C09115=1110.868,346.804,-84.343,-177.299,10.930,149.499
C09116=1110.872,346.556,-84.309,-177.302,10.928,149.499
C09117=1110.876,346.309,-84.274,-177.305,10.925,149.499
C09118=1110.880,346.062,-84.238,-177.308,10.923,149.499
C09119=1110.883,345.813,-84.203,-177.312,10.920,149.500
C09120=1110.888,345.567,-84.168,-177.314,10.918,149.500
C09121=1110.892,345.318,-84.133,-177.317,10.916,149.500
C09122=1110.895,345.071,-84.098,-177.321,10.913,149.500
C09123=1110.899,344.824,-84.064,-177.324,10.911,149.500
C09124=1110.903,344.576,-84.028,-177.327,10.908,149.501
C09125=1110.907,344.328,-83.994,-177.330,10.906,149.501
C09126=1110.911,344.081,-83.959,-177.334,10.903,149.501
C09127=1110.914,343.834,-83.924,-177.337,10.901,149.501
C09128=1110.919,343.586,-83.890,-177.340,10.898,149.501
C09129=1110.923,343.339,-83.854,-177.343,10.897,149.502
C09130=1110.927,343.091,-83.819,-177.346,10.894,149.502
C09131=1110.930,342.843,-83.785,-177.349,10.891,149.502
C09132=1110.934,342.596,-83.750,-177.352,10.889,149.502
C09133=1110.939,342.349,-83.715,-177.356,10.886,149.502
C09134=1110.943,342.100,-83.681,-177.359,10.884,149.503
C09135=1110.945,341.853,-83.646,-177.362,10.881,149.503
C09136=1110.950,341.606,-83.611,-177.365,10.879,149.503
C09137=1110.954,341.358,-83.576,-177.369,10.876,149.503
C09138=1110.958,341.111,-83.543,-177.372,10.874,149.503
C09139=1110.962,340.863,-83.507,-177.374,10.872,149.503
C09140=1110.966,340.616,-83.473,-177.378,10.869,149.504
C09141=1110.969,340.368,-83.438,-177.381,10.867,149.504
C09142=1110.974,340.120,-83.404,-177.384,10.864,149.504
C09143=1110.978,339.873,-83.368,-177.387,10.862,149.504
C09144=1110.981,339.625,-83.334,-177.390,10.859,149.504
C09145=1110.985,339.378,-83.300,-177.394,10.857,149.505
C09146=1110.989,339.130,-83.265,-177.397,10.854,149.505
C09147=1110.993,338.882,-83.231,-177.400,10.852,149.505
C09148=1110.997,338.634,-83.196,-177.403,10.849,149.505
C09149=1111.002,338.387,-83.162,-177.407,10.847,149.505
C09150=1111.005,338.139,-83.127,-177.409,10.845,149.506
C09151=1111.009,337.892,-83.092,-177.413,10.842,149.506
C09152=1111.012,337.645,-83.058,-177.415,10.840,149.506
C09153=1111.016,337.433,-83.029,-177.419,10.837,149.506
C09154=1111.019,337.221,-82.999,-177.421,10.835,149.506
C09155=1111.023,337.009,-82.970,-177.424,10.833,149.507
C09156=1111.026,336.797,-82.940,-177.427,10.831,149.507
C09157=1111.030,336.585,-82.911,-177.429,10.829,149.507
C09158=1111.034,336.373,-82.881,-177.432,10.827,149.507
C09159=1111.037,336.161,-82.852,-177.435,10.825,149.507
C09160=1111.039,335.949,-82.823,-177.437,10.823,149.507
C09161=1111.044,335.702,-82.788,-177.441,10.820,149.508
C09162=1111.047,335.454,-82.754,-177.444,10.818,149.508
C09163=1111.052,335.206,-82.720,-177.447,10.815,149.508
C09164=1111.056,334.959,-82.686,-177.450,10.812,149.508
C09165=1111.060,334.710,-82.652,-177.453,10.811,149.508
C09166=1111.063,334.463,-82.618,-177.456,10.808,149.509
C09167=1111.067,334.215,-82.583,-177.459,10.806,149.509
C09168=1111.071,333.968,-82.549,-177.462,10.803,149.509
C09169=1111.075,333.720,-82.515,-177.466,10.801,149.509
C09170=1111.079,333.473,-82.480,-177.469,10.798,149.509
C09171=1111.083,333.225,-82.447,-177.472,10.795,149.509
C09172=1111.087,332.977,-82.412,-177.475,10.793,149.510
C09173=1111.091,332.730,-82.379,-177.479,10.790,149.510
C09174=1111.094,332.482,-82.344,-177.481,10.788,149.510
C09175=1111.099,332.234,-82.311,-177.484,10.786,149.510
C09176=1111.103,331.987,-82.277,-177.487,10.784,149.510
C09177=1111.106,331.739,-82.242,-177.490,10.781,149.510
C09178=1111.111,331.492,-82.208,-177.494,10.778,149.511
C09179=1111.115,331.244,-82.175,-177.497,10.776,149.511
C09180=1111.118,330.996,-82.141,-177.500,10.773,149.511
C09181=1111.123,330.749,-82.106,-177.503,10.771,149.511
C09182=1111.127,330.501,-82.073,-177.507,10.768,149.512
C09183=1111.130,330.253,-82.039,-177.510,10.766,149.512
C09184=1111.134,330.006,-82.005,-177.513,10.763,149.512
C09185=1111.139,329.758,-81.971,-177.516,10.761,149.512
C09186=1111.142,329.510,-81.937,-177.519,10.759,149.512
C09187=1111.146,329.263,-81.904,-177.522,10.756,149.512
C09188=1111.150,329.015,-81.870,-177.525,10.754,149.513
C09189=1111.154,328.767,-81.836,-177.528,10.751,149.513
C09190=1111.158,328.520,-81.802,-177.531,10.748,149.513
C09191=1111.162,328.272,-81.768,-177.535,10.746,149.513
C09192=1111.165,328.024,-81.734,-177.538,10.743,149.513
C09193=1111.170,327.777,-81.700,-177.541,10.741,149.513
C09194=1111.174,327.529,-81.667,-177.544,10.738,149.514
C09195=1111.178,327.282,-81.633,-177.547,10.737,149.514
C09196=1111.182,327.033,-81.599,-177.550,10.734,149.514
C09197=1111.186,326.786,-81.566,-177.553,10.731,149.514
C09198=1111.190,326.539,-81.532,-177.556,10.729,149.515
C09199=1111.194,326.290,-81.499,-177.559,10.726,149.515
C09200=1111.198,326.043,-81.464,-177.563,10.724,149.515
C09201=1111.202,325.795,-81.431,-177.566,10.721,149.515
C09202=1111.206,325.547,-81.398,-177.569,10.718,149.515
C09203=1111.210,325.300,-81.364,-177.572,10.716,149.515
C09204=1111.213,325.052,-81.331,-177.576,10.714,149.516
C09205=1111.217,324.804,-81.298,-177.578,10.712,149.516
C09206=1111.221,324.557,-81.264,-177.581,10.709,149.516
C09207=1111.225,324.309,-81.231,-177.585,10.707,149.516
C09208=1111.230,324.061,-81.197,-177.587,10.704,149.516
C09209=1111.233,323.849,-81.168,-177.591,10.701,149.517
C09210=1111.237,323.637,-81.139,-177.593,10.699,149.517
C09211=1111.240,323.424,-81.111,-177.596,10.698,149.517
C09212=1111.243,323.213,-81.082,-177.599,10.695,149.517
C09213=1111.246,323.000,-81.053,-177.601,10.693,149.517
C09214=1111.250,322.788,-81.025,-177.604,10.691,149.517
C09215=1111.253,322.577,-80.996,-177.607,10.689,149.517
C09216=1111.256,322.364,-80.968,-177.609,10.687,149.518
C09217=1111.260,322.117,-80.935,-177.612,10.684,149.518
C09218=1111.264,321.869,-80.902,-177.616,10.682,149.518
C09219=1111.269,321.621,-80.869,-177.618,10.679,149.518
C09220=1111.272,321.374,-80.835,-177.621,10.677,149.518
C09221=1111.276,321.126,-80.801,-177.624,10.675,149.519
C09222=1111.280,320.878,-80.768,-177.627,10.672,149.519
C09223=1111.284,320.630,-80.735,-177.631,10.670,149.519
C09224=1111.288,320.382,-80.702,-177.634,10.667,149.519
C09225=1111.293,320.135,-80.668,-177.637,10.664,149.519
C09226=1111.297,319.887,-80.635,-177.640,10.662,149.519
C09227=1111.301,319.639,-80.602,-177.643,10.659,149.520
C09228=1111.304,319.391,-80.569,-177.647,10.657,149.520
C09229=1111.308,319.143,-80.536,-177.650,10.654,149.520
C09230=1111.312,318.896,-80.503,-177.652,10.652,149.520
C09231=1111.316,318.648,-80.470,-177.656,10.650,149.520
C09232=1111.320,318.400,-80.437,-177.658,10.647,149.520
C09233=1111.324,318.152,-80.403,-177.662,10.645,149.521
C09234=1111.328,317.905,-80.370,-177.665,10.642,149.521
C09235=1111.333,317.657,-80.337,-177.668,10.639,149.521
C09236=1111.336,317.410,-80.305,-177.671,10.637,149.521
C09237=1111.340,317.162,-80.271,-177.674,10.634,149.521
C09238=1111.344,316.914,-80.238,-177.678,10.632,149.522
C09239=1111.348,316.666,-80.205,-177.681,10.629,149.522
C09240=1111.353,316.418,-80.173,-177.683,10.627,149.522
C09241=1111.356,316.171,-80.140,-177.687,10.625,149.522
C09242=1111.360,315.922,-80.107,-177.689,10.622,149.522
C09243=1111.364,315.674,-80.073,-177.693,10.620,149.522
C09244=1111.368,315.427,-80.040,-177.696,10.617,149.523
C09245=1111.372,315.178,-80.008,-177.699,10.614,149.523
C09246=1111.376,314.931,-79.975,-177.702,10.612,149.523
C09247=1111.380,314.683,-79.942,-177.705,10.609,149.523
C09248=1111.384,314.436,-79.909,-177.709,10.607,149.523
C09249=1111.388,314.187,-79.877,-177.712,10.604,149.524
C09250=1111.392,313.940,-79.844,-177.714,10.602,149.524
C09251=1111.396,313.692,-79.811,-177.718,10.600,149.524
C09252=1111.400,313.444,-79.778,-177.720,10.597,149.524
C09253=1111.404,313.196,-79.746,-177.724,10.595,149.524
C09254=1111.408,312.949,-79.713,-177.727,10.592,149.524
C09255=1111.413,312.701,-79.681,-177.730,10.589,149.525
C09256=1111.417,312.453,-79.648,-177.733,10.587,149.525
C09257=1111.421,312.206,-79.615,-177.736,10.584,149.525
C09258=1111.424,311.958,-79.583,-177.740,10.582,149.525
C09259=1111.429,311.710,-79.550,-177.743,10.579,149.525
C09260=1111.433,311.462,-79.517,-177.745,10.577,149.526
C09261=1111.436,311.214,-79.485,-177.748,10.575,149.526
C09262=1111.441,310.966,-79.452,-177.752,10.572,149.526
C09263=1111.445,310.718,-79.419,-177.754,10.569,149.526
C09264=1111.448,310.471,-79.387,-177.758,10.567,149.526
C09265=1111.452,310.258,-79.360,-177.760,10.565,149.526
C09266=1111.455,310.046,-79.332,-177.763,10.562,149.527
C09267=1111.460,309.834,-79.303,-177.766,10.560,149.527
C09268=1111.463,309.621,-79.276,-177.768,10.558,149.527
C09269=1111.466,309.409,-79.248,-177.771,10.556,149.527
C09270=1111.469,309.197,-79.220,-177.774,10.554,149.527
C09271=1111.473,308.985,-79.192,-177.776,10.552,149.527
C09272=1111.476,308.773,-79.165,-177.779,10.550,149.528
C09273=1111.481,308.525,-79.132,-177.782,10.547,149.528
C09274=1111.484,308.277,-79.100,-177.786,10.544,149.528
C09275=1111.489,308.029,-79.067,-177.788,10.542,149.528
C09276=1111.492,307.781,-79.035,-177.791,10.540,149.528
C09277=1111.497,307.533,-79.002,-177.794,10.537,149.528
C09278=1111.501,307.286,-78.971,-177.797,10.535,149.529
C09279=1111.505,307.037,-78.938,-177.800,10.532,149.529
C09280=1111.509,306.790,-78.906,-177.804,10.530,149.529
C09281=1111.512,306.542,-78.874,-177.807,10.527,149.529
C09282=1111.517,306.294,-78.841,-177.810,10.524,149.529
C09283=1111.521,306.046,-78.810,-177.813,10.522,149.529
C09284=1111.525,305.798,-78.777,-177.816,10.520,149.530
C09285=1111.529,305.550,-78.745,-177.819,10.517,149.530
C09286=1111.534,305.302,-78.712,-177.822,10.515,149.530
C09287=1111.537,305.054,-78.681,-177.825,10.512,149.530
C09288=1111.541,304.807,-78.648,-177.828,10.510,149.530
C09289=1111.546,304.559,-78.616,-177.831,10.507,149.531
C09290=1111.549,304.311,-78.584,-177.834,10.504,149.531
C09291=1111.554,304.063,-78.552,-177.838,10.502,149.531
C09292=1111.558,303.815,-78.520,-177.841,10.499,149.531
C09293=1111.562,303.567,-78.488,-177.844,10.497,149.531
C09294=1111.566,303.319,-78.456,-177.846,10.495,149.531
C09295=1111.570,303.071,-78.424,-177.850,10.492,149.532
C09296=1111.574,302.824,-78.392,-177.852,10.489,149.532
C09297=1111.578,302.576,-78.359,-177.856,10.487,149.532
C09298=1111.582,302.328,-78.328,-177.859,10.484,149.532
C09299=1111.586,302.080,-78.296,-177.862,10.482,149.532
C09300=1111.591,301.832,-78.264,-177.865,10.479,149.532
C09301=1111.595,301.584,-78.232,-177.868,10.477,149.533
C09302=1111.598,301.336,-78.200,-177.871,10.474,149.533
C09303=1111.603,301.088,-78.168,-177.874,10.472,149.533
C09304=1111.607,300.840,-78.136,-177.877,10.469,149.533
C09305=1111.611,300.592,-78.104,-177.880,10.467,149.533
C09306=1111.615,300.345,-78.073,-177.883,10.464,149.533
C09307=1111.620,300.096,-78.041,-177.887,10.462,149.534
C09308=1111.624,299.848,-78.009,-177.889,10.459,149.534
C09309=1111.628,299.601,-77.978,-177.893,10.457,149.534
C09310=1111.632,299.353,-77.946,-177.896,10.454,149.534
C09311=1111.635,299.104,-77.914,-177.899,10.451,149.534
C09312=1111.640,298.857,-77.882,-177.902,10.449,149.534
C09313=1111.644,298.609,-77.850,-177.905,10.447,149.535
C09314=1111.648,298.361,-77.818,-177.908,10.444,149.535
C09315=1111.652,298.113,-77.787,-177.911,10.442,149.535
C09316=1111.656,297.865,-77.756,-177.914,10.439,149.535
C09317=1111.660,297.617,-77.724,-177.917,10.437,149.535
C09318=1111.665,297.369,-77.692,-177.920,10.434,149.535
C09319=1111.669,297.120,-77.661,-177.923,10.431,149.536
C09320=1111.673,296.872,-77.629,-177.926,10.429,149.536
C09321=1111.676,296.660,-77.601,-177.929,10.427,149.536
C09322=1111.680,296.448,-77.575,-177.931,10.425,149.536
C09323=1111.683,296.236,-77.548,-177.934,10.422,149.536
C09324=1111.687,296.023,-77.521,-177.937,10.420,149.536
C09325=1111.690,295.811,-77.494,-177.939,10.418,149.537
C09326=1111.694,295.599,-77.467,-177.942,10.416,149.537
C09327=1111.697,295.386,-77.440,-177.945,10.414,149.537
C09328=1111.700,295.174,-77.413,-177.947,10.412,149.537
C09329=1111.705,294.926,-77.381,-177.950,10.409,149.537
C09330=1111.709,294.678,-77.350,-177.953,10.407,149.537
C09331=1111.713,294.430,-77.318,-177.956,10.404,149.538
C09332=1111.718,294.182,-77.287,-177.959,10.401,149.538
C09333=1111.721,293.934,-77.256,-177.963,10.399,149.538
C09334=1111.725,293.686,-77.224,-177.966,10.396,149.538
C09335=1111.730,293.438,-77.193,-177.969,10.394,149.538
C09336=1111.733,293.190,-77.162,-177.971,10.392,149.538
C09337=1111.737,292.942,-77.131,-177.974,10.389,149.539
C09338=1111.741,292.694,-77.099,-177.978,10.387,149.539
C09339=1111.746,292.446,-77.068,-177.981,10.384,149.539
C09340=1111.749,292.198,-77.036,-177.984,10.381,149.539
C09341=1111.754,291.950,-77.006,-177.987,10.379,149.539
C09342=1111.758,291.702,-76.974,-177.990,10.376,149.540
C09343=1111.762,291.454,-76.943,-177.993,10.373,149.540
C09344=1111.766,291.206,-76.911,-177.996,10.372,149.540
C09345=1111.771,290.958,-76.880,-177.999,10.369,149.540
C09346=1111.775,290.709,-76.849,-178.002,10.367,149.540
C09347=1111.779,290.462,-76.818,-178.005,10.364,149.540
C09348=1111.782,290.214,-76.787,-178.008,10.361,149.540
C09349=1111.787,289.966,-76.756,-178.011,10.359,149.541
C09350=1111.791,289.718,-76.725,-178.014,10.356,149.541
C09351=1111.795,289.470,-76.694,-178.018,10.354,149.541
C09352=1111.799,289.222,-76.662,-178.020,10.351,149.541
C09353=1111.804,288.974,-76.631,-178.023,10.349,149.542
C09354=1111.807,288.726,-76.601,-178.026,10.346,149.542
C09355=1111.811,288.478,-76.570,-178.029,10.344,149.542
C09356=1111.816,288.230,-76.539,-178.032,10.341,149.542
C09357=1111.820,287.982,-76.507,-178.035,10.338,149.542
C09358=1111.824,287.734,-76.477,-178.039,10.336,149.542
C09359=1111.828,287.485,-76.446,-178.042,10.333,149.542
C09360=1111.832,287.238,-76.415,-178.045,10.331,149.543
C09361=1111.836,286.989,-76.384,-178.048,10.328,149.543
C09362=1111.841,286.741,-76.353,-178.051,10.326,149.543
C09363=1111.844,286.494,-76.323,-178.053,10.324,149.543
C09364=1111.848,286.245,-76.291,-178.056,10.321,149.543
C09365=1111.853,285.997,-76.261,-178.060,10.318,149.544
C09366=1111.857,285.750,-76.229,-178.063,10.316,149.544
C09367=1111.861,285.501,-76.199,-178.066,10.313,149.544
C09368=1111.865,285.253,-76.168,-178.069,10.310,149.544
C09369=1111.869,285.005,-76.137,-178.072,10.308,149.544
C09370=1111.873,284.757,-76.107,-178.075,10.306,149.544
C09371=1111.878,284.509,-76.076,-178.078,10.303,149.544
C09372=1111.882,284.260,-76.045,-178.081,10.301,149.545
C09373=1111.886,284.013,-76.014,-178.084,10.298,149.545
C09374=1111.890,283.765,-75.984,-178.087,10.296,149.545
C09375=1111.894,283.516,-75.953,-178.090,10.293,149.545
C09376=1111.898,283.269,-75.922,-178.093,10.290,149.545
C09377=1111.902,283.055,-75.896,-178.096,10.289,149.546
C09378=1111.906,282.844,-75.870,-178.098,10.287,149.546
C09379=1111.909,282.631,-75.844,-178.101,10.284,149.546
C09380=1111.913,282.418,-75.817,-178.103,10.282,149.546
C09381=1111.916,282.206,-75.791,-178.106,10.280,149.546
C09382=1111.920,281.994,-75.765,-178.109,10.277,149.546
C09383=1111.924,281.781,-75.739,-178.111,10.275,149.546
C09384=1111.927,281.568,-75.713,-178.114,10.273,149.547
C09385=1111.932,281.320,-75.682,-178.117,10.271,149.547
C09386=1111.935,281.072,-75.652,-178.120,10.268,149.547
C09387=1111.939,280.824,-75.621,-178.123,10.265,149.547
C09388=1111.943,280.576,-75.591,-178.126,10.263,149.547
C09389=1111.948,280.328,-75.560,-178.129,10.260,149.547
C09390=1111.952,280.080,-75.530,-178.132,10.258,149.548
C09391=1111.956,279.831,-75.499,-178.135,10.255,149.548
C09392=1111.960,279.584,-75.469,-178.138,10.252,149.548
C09393=1111.965,279.336,-75.438,-178.142,10.250,149.548
C09394=1111.969,279.087,-75.409,-178.145,10.247,149.548
C09395=1111.973,278.839,-75.378,-178.147,10.244,149.548
C09396=1111.977,278.591,-75.348,-178.151,10.242,149.549
C09397=1111.981,278.343,-75.317,-178.154,10.239,149.549
C09398=1111.986,278.095,-75.287,-178.157,10.236,149.549
C09399=1111.990,277.847,-75.257,-178.159,10.234,149.549
C09400=1111.993,277.598,-75.226,-178.162,10.232,149.549
C09401=1111.998,277.350,-75.197,-178.165,10.229,149.549
C09402=1112.002,277.102,-75.166,-178.168,10.227,149.549
C09403=1112.006,276.855,-75.136,-178.171,10.224,149.550
C09404=1112.011,276.606,-75.106,-178.174,10.221,149.550
C09405=1112.014,276.358,-75.075,-178.177,10.219,149.550
C09406=1112.018,276.109,-75.046,-178.180,10.216,149.550
C09407=1112.023,275.861,-75.015,-178.183,10.213,149.550
C09408=1112.027,275.614,-74.985,-178.186,10.210,149.550
C09409=1112.031,275.366,-74.955,-178.189,10.208,149.550
C09410=1112.036,275.118,-74.924,-178.192,10.205,149.550
C09411=1112.039,274.869,-74.895,-178.195,10.203,149.551
C09412=1112.043,274.621,-74.864,-178.198,10.200,149.551
C09413=1112.048,274.372,-74.834,-178.201,10.198,149.551
C09414=1112.052,274.125,-74.804,-178.204,10.195,149.551
C09415=1112.056,273.876,-74.775,-178.207,10.192,149.551
C09416=1112.061,273.628,-74.744,-178.209,10.189,149.551
C09417=1112.065,273.380,-74.715,-178.212,10.187,149.551
C09418=1112.069,273.132,-74.685,-178.215,10.184,149.551
C09419=1112.073,272.884,-74.655,-178.218,10.182,149.551
C09420=1112.077,272.635,-74.625,-178.221,10.179,149.552
C09421=1112.081,272.387,-74.594,-178.224,10.177,149.552
C09422=1112.085,272.139,-74.565,-178.227,10.174,149.552
C09423=1112.090,271.891,-74.535,-178.230,10.171,149.552
C09424=1112.094,271.643,-74.505,-178.233,10.168,149.552
C09425=1112.098,271.395,-74.475,-178.236,10.166,149.552
C09426=1112.103,271.146,-74.446,-178.238,10.164,149.552
C09427=1112.106,270.899,-74.416,-178.241,10.161,149.552
C09428=1112.111,270.650,-74.386,-178.244,10.158,149.553
C09429=1112.116,270.402,-74.356,-178.247,10.155,149.553
C09430=1112.120,270.154,-74.327,-178.250,10.153,149.553
C09431=1112.124,269.906,-74.297,-178.252,10.151,149.553
C09432=1112.128,269.658,-74.267,-178.255,10.148,149.553
C09433=1112.131,269.445,-74.241,-178.257,10.146,149.553
C09434=1112.135,269.232,-74.216,-178.260,10.143,149.553
C09435=1112.138,269.019,-74.190,-178.263,10.141,149.553
C09436=1112.143,268.807,-74.166,-178.265,10.139,149.553
C09437=1112.146,268.594,-74.140,-178.267,10.137,149.553
C09438=1112.150,268.382,-74.114,-178.270,10.134,149.554
C09439=1112.153,268.168,-74.089,-178.272,10.132,149.554
C09440=1112.157,267.956,-74.064,-178.274,10.130,149.554
C09441=1112.161,267.708,-74.034,-178.277,10.127,149.554
C09442=1112.165,267.460,-74.005,-178.280,10.125,149.554
C09443=1112.170,267.211,-73.975,-178.282,10.123,149.554
C09444=1112.174,266.963,-73.946,-178.285,10.120,149.554
C09445=1112.178,266.715,-73.916,-178.288,10.117,149.554
C09446=1112.182,266.467,-73.886,-178.291,10.115,149.554
C09447=1112.186,266.219,-73.857,-178.294,10.112,149.555
C09448=1112.190,265.971,-73.827,-178.297,10.110,149.555
C09449=1112.194,265.723,-73.798,-178.299,10.107,149.555
C09450=1112.199,265.474,-73.768,-178.302,10.105,149.555
C09451=1112.203,265.226,-73.739,-178.305,10.102,149.555
C09452=1112.207,264.978,-73.709,-178.308,10.100,149.555
C09453=1112.211,264.729,-73.680,-178.310,10.098,149.555
C09454=1112.215,264.481,-73.650,-178.313,10.095,149.555
C09455=1112.220,264.232,-73.622,-178.316,10.092,149.556
C09456=1112.224,263.984,-73.592,-178.319,10.089,149.556
C09457=1112.229,263.736,-73.563,-178.323,10.087,149.556
C09458=1112.233,263.488,-73.534,-178.326,10.084,149.556
C09459=1112.237,263.240,-73.504,-178.328,10.081,149.556
C09460=1112.241,262.992,-73.475,-178.331,10.079,149.556
C09461=1112.246,262.743,-73.445,-178.334,10.076,149.556
C09462=1112.250,262.495,-73.416,-178.338,10.074,149.557
C09463=1112.254,262.247,-73.386,-178.341,10.071,149.557
C09464=1112.258,261.998,-73.358,-178.344,10.068,149.557
C09465=1112.262,261.751,-73.329,-178.346,10.065,149.557
C09466=1112.267,261.502,-73.300,-178.349,10.063,149.557
C09467=1112.271,261.254,-73.270,-178.352,10.060,149.557
C09468=1112.275,261.006,-73.241,-178.355,10.057,149.557
C09469=1112.279,260.757,-73.212,-178.358,10.054,149.557
C09470=1112.284,260.509,-73.183,-178.361,10.051,149.558
C09471=1112.288,260.261,-73.154,-178.364,10.049,149.558
C09472=1112.292,260.013,-73.125,-178.367,10.046,149.558
C09473=1112.296,259.764,-73.096,-178.370,10.043,149.558
C09474=1112.301,259.516,-73.067,-178.373,10.040,149.558
C09475=1112.305,259.267,-73.038,-178.375,10.037,149.558
C09476=1112.309,259.019,-73.008,-178.378,10.035,149.558
C09477=1112.313,258.772,-72.980,-178.381,10.032,149.558
C09478=1112.318,258.523,-72.951,-178.384,10.029,149.558
C09479=1112.322,258.275,-72.922,-178.387,10.026,149.558
C09480=1112.326,258.026,-72.892,-178.390,10.023,149.558
C09481=1112.330,257.778,-72.864,-178.393,10.020,149.558
C09482=1112.335,257.530,-72.835,-178.396,10.018,149.558
C09483=1112.339,257.281,-72.806,-178.398,10.016,149.559
C09484=1112.343,257.033,-72.777,-178.400,10.013,149.558
C09485=1112.347,256.784,-72.749,-178.403,10.010,149.559
C09486=1112.352,256.537,-72.720,-178.406,10.007,149.559
C09487=1112.356,256.288,-72.691,-178.409,10.004,149.559
C09488=1112.360,256.040,-72.662,-178.412,10.001,149.559
C09489=1112.364,255.827,-72.637,-178.413,10.000,149.559
C09490=1112.367,255.615,-72.613,-178.415,9.997,149.559
C09491=1112.371,255.401,-72.588,-178.417,9.996,149.559
C09492=1112.375,255.189,-72.563,-178.419,9.994,149.559
C09493=1112.379,254.976,-72.539,-178.420,9.992,149.559
C09494=1112.382,254.763,-72.514,-178.422,9.990,149.559
C09495=1112.386,254.551,-72.489,-178.424,9.988,149.559
C09496=1112.390,254.338,-72.464,-178.426,9.987,149.559
C09497=1112.393,254.089,-72.436,-178.429,9.984,149.559
C09498=1112.398,253.841,-72.407,-178.431,9.982,149.559
C09499=1112.403,253.593,-72.379,-178.433,9.980,149.559
C09500=1112.406,253.344,-72.350,-178.436,9.977,149.559
C09501=1112.411,253.096,-72.321,-178.438,9.975,149.559
C09502=1112.415,252.848,-72.293,-178.440,9.973,149.559
C09503=1112.419,252.599,-72.264,-178.444,9.971,149.560
C09504=1112.424,252.351,-72.235,-178.447,9.968,149.560
C09505=1112.428,252.103,-72.207,-178.449,9.966,149.560
C09506=1112.432,251.854,-72.178,-178.452,9.963,149.560
C09507=1112.436,251.606,-72.150,-178.455,9.961,149.560
C09508=1112.441,251.358,-72.121,-178.458,9.958,149.561
C09509=1112.445,251.109,-72.093,-178.461,9.955,149.561
C09510=1112.449,250.861,-72.064,-178.465,9.953,149.561
C09511=1112.453,250.613,-72.036,-178.467,9.950,149.561
C09512=1112.458,250.364,-72.007,-178.471,9.948,149.561
C09513=1112.462,250.116,-71.979,-178.474,9.945,149.561
C09514=1112.467,249.868,-71.951,-178.477,9.941,149.562
C09515=1112.470,249.620,-71.922,-178.481,9.939,149.562
C09516=1112.475,249.371,-71.893,-178.484,9.935,149.562
C09517=1112.479,249.123,-71.865,-178.488,9.933,149.562
C09518=1112.483,248.874,-71.836,-178.491,9.929,149.562
C09519=1112.488,248.626,-71.809,-178.495,9.926,149.563
C09520=1112.491,248.378,-71.781,-178.499,9.923,149.563
C09521=1112.497,248.129,-71.752,-178.502,9.919,149.563
C09522=1112.500,247.881,-71.724,-178.506,9.916,149.563
C09523=1112.505,247.633,-71.696,-178.510,9.913,149.563
C09524=1112.509,247.384,-71.668,-178.512,9.909,149.563
C09525=1112.513,247.135,-71.639,-178.515,9.906,149.563
C09526=1112.518,246.887,-71.611,-178.517,9.904,149.563
C09527=1112.522,246.639,-71.583,-178.519,9.901,149.563
C09528=1112.526,246.391,-71.555,-178.521,9.899,149.563
C09529=1112.531,246.142,-71.526,-178.524,9.896,149.563
C09530=1112.535,245.894,-71.499,-178.526,9.893,149.563
C09531=1112.539,245.645,-71.470,-178.529,9.890,149.563
C09532=1112.544,245.397,-71.442,-178.531,9.888,149.563
C09533=1112.548,245.149,-71.414,-178.533,9.885,149.563
C09534=1112.552,244.901,-71.386,-178.535,9.883,149.563
C09535=1112.556,244.652,-71.357,-178.538,9.880,149.563
C09536=1112.561,244.404,-71.330,-178.540,9.877,149.563
C09537=1112.564,244.156,-71.301,-178.543,9.875,149.563
C09538=1112.570,243.907,-71.274,-178.545,9.872,149.563
C09539=1112.574,243.658,-71.246,-178.547,9.869,149.563
C09540=1112.578,243.410,-71.218,-178.549,9.867,149.563
C09541=1112.582,243.162,-71.190,-178.552,9.864,149.563
C09542=1112.587,242.913,-71.161,-178.554,9.862,149.563
C09543=1112.591,242.665,-71.133,-178.557,9.859,149.563
C09544=1112.595,242.416,-71.106,-178.559,9.857,149.563
C09545=1112.599,242.204,-71.082,-178.561,9.855,149.563
C09546=1112.602,241.991,-71.058,-178.563,9.853,149.563
C09547=1112.607,241.778,-71.034,-178.565,9.850,149.563
C09548=1112.610,241.565,-71.010,-178.568,9.849,149.563
C09549=1112.613,241.352,-70.986,-178.570,9.845,149.563
C09550=1112.617,241.139,-70.962,-178.572,9.843,149.563
C09551=1112.621,240.926,-70.939,-178.574,9.841,149.563
C09552=1112.624,240.713,-70.915,-178.577,9.839,149.563
C09553=1112.629,240.465,-70.887,-178.579,9.837,149.563
C09554=1112.633,240.216,-70.859,-178.581,9.834,149.563
C09555=1112.638,239.968,-70.831,-178.584,9.831,149.563
C09556=1112.642,239.720,-70.804,-178.587,9.829,149.564
C09557=1112.646,239.471,-70.776,-178.589,9.826,149.563
C09558=1112.651,239.223,-70.748,-178.592,9.824,149.564
C09559=1112.654,238.974,-70.720,-178.595,9.821,149.564
C09560=1112.660,238.726,-70.693,-178.597,9.819,149.564
C09561=1112.664,238.478,-70.665,-178.599,9.816,149.564
C09562=1112.668,238.229,-70.637,-178.602,9.814,149.564
C09563=1112.672,237.981,-70.610,-178.605,9.811,149.564
C09564=1112.677,237.733,-70.582,-178.608,9.809,149.564
C09565=1112.681,237.483,-70.554,-178.610,9.806,149.564
C09566=1112.685,237.236,-70.527,-178.613,9.803,149.564
C09567=1112.689,236.986,-70.499,-178.615,9.801,149.564
C09568=1112.694,236.739,-70.472,-178.618,9.798,149.564
C09569=1112.698,236.490,-70.444,-178.621,9.796,149.565
C09570=1112.702,236.241,-70.416,-178.624,9.792,149.565
C09571=1112.707,235.993,-70.389,-178.626,9.790,149.565
C09572=1112.711,235.745,-70.361,-178.629,9.788,149.565
C09573=1112.716,235.497,-70.334,-178.632,9.785,149.565
C09574=1112.719,235.248,-70.306,-178.635,9.782,149.565
C09575=1112.724,235.000,-70.279,-178.637,9.780,149.565
C09576=1112.729,234.751,-70.252,-178.640,9.777,149.565
C09577=1112.732,234.502,-70.224,-178.643,9.774,149.565
C09578=1112.737,234.254,-70.197,-178.646,9.772,149.565
C09579=1112.742,234.005,-70.170,-178.649,9.769,149.565
C09580=1112.746,233.757,-70.142,-178.652,9.766,149.566
C09581=1112.750,233.508,-70.115,-178.654,9.763,149.566
C09582=1112.755,233.261,-70.087,-178.656,9.761,149.566
C09583=1112.759,233.012,-70.060,-178.659,9.758,149.566
C09584=1112.763,232.763,-70.032,-178.662,9.756,149.566
C09585=1112.768,232.514,-70.005,-178.665,9.752,149.566
C09586=1112.772,232.267,-69.978,-178.668,9.750,149.566
C09587=1112.776,232.018,-69.951,-178.671,9.747,149.566
C09588=1112.780,231.769,-69.924,-178.674,9.744,149.566
C09589=1112.785,231.521,-69.897,-178.676,9.741,149.566
C09590=1112.789,231.273,-69.869,-178.679,9.738,149.566
C09591=1112.794,231.024,-69.842,-178.682,9.736,149.566
C09592=1112.798,230.775,-69.814,-178.685,9.733,149.566
C09593=1112.802,230.527,-69.788,-178.688,9.730,149.566
C09594=1112.807,230.278,-69.761,-178.690,9.727,149.567
C09595=1112.811,230.030,-69.734,-178.693,9.724,149.567
C09596=1112.816,229.782,-69.706,-178.696,9.721,149.567
C09597=1112.820,229.533,-69.679,-178.700,9.718,149.567
C09598=1112.824,229.285,-69.652,-178.702,9.715,149.567
C09599=1112.828,229.036,-69.625,-178.705,9.712,149.567
C09600=1112.833,228.788,-69.598,-178.708,9.709,149.567
C09601=1112.837,228.575,-69.574,-178.710,9.707,149.567
C09602=1112.841,228.361,-69.552,-178.712,9.704,149.567
C09603=1112.844,228.148,-69.529,-178.715,9.702,149.567
C09604=1112.847,227.935,-69.505,-178.717,9.698,149.567
C09605=1112.852,227.723,-69.482,-178.719,9.696,149.567
C09606=1112.856,227.509,-69.459,-178.722,9.693,149.567
C09607=1112.859,227.296,-69.436,-178.724,9.691,149.567
C09608=1112.862,227.084,-69.413,-178.726,9.688,149.567
C09609=1112.867,226.835,-69.386,-178.729,9.685,149.567
C09610=1112.872,226.587,-69.359,-178.732,9.682,149.567
C09611=1112.876,226.338,-69.332,-178.734,9.679,149.567
C09612=1112.880,226.089,-69.306,-178.737,9.676,149.567
C09613=1112.885,225.840,-69.279,-178.739,9.673,149.567
C09614=1112.889,225.592,-69.252,-178.742,9.670,149.567
C09615=1112.893,225.343,-69.225,-178.745,9.667,149.567
C09616=1112.898,225.095,-69.198,-178.747,9.664,149.567
C09617=1112.902,224.847,-69.171,-178.750,9.661,149.567
C09618=1112.906,224.598,-69.144,-178.753,9.658,149.567
C09619=1112.911,224.350,-69.117,-178.755,9.654,149.566
C09620=1112.915,224.101,-69.092,-178.758,9.651,149.566
C09621=1112.920,223.852,-69.065,-178.760,9.648,149.566
C09622=1112.924,223.604,-69.038,-178.763,9.645,149.566
C09623=1112.929,223.356,-69.011,-178.765,9.642,149.566
C09624=1112.933,223.108,-68.985,-178.768,9.639,149.566
C09625=1112.937,222.858,-68.958,-178.770,9.636,149.566
C09626=1112.942,222.609,-68.931,-178.773,9.633,149.566
C09627=1112.945,222.361,-68.904,-178.775,9.630,149.566
C09628=1112.950,222.113,-68.877,-178.778,9.626,149.566
C09629=1112.954,221.864,-68.852,-178.780,9.623,149.566
C09630=1112.959,221.615,-68.824,-178.783,9.620,149.566
C09631=1112.963,221.367,-68.798,-178.785,9.617,149.566
C09632=1112.968,221.118,-68.772,-178.788,9.614,149.566
C09633=1112.972,220.870,-68.745,-178.790,9.611,149.566
C09634=1112.976,220.621,-68.718,-178.793,9.608,149.565
C09635=1112.981,220.372,-68.692,-178.795,9.604,149.565
C09636=1112.985,220.124,-68.665,-178.798,9.601,149.565
C09637=1112.990,219.875,-68.640,-178.799,9.599,149.565
C09638=1112.994,219.627,-68.612,-178.802,9.596,149.565
C09639=1112.998,219.378,-68.586,-178.805,9.593,149.565
C09640=1113.003,219.130,-68.561,-178.807,9.590,149.565
C09641=1113.008,218.882,-68.534,-178.809,9.586,149.565
C09642=1113.012,218.633,-68.508,-178.812,9.583,149.565
C09643=1113.017,218.385,-68.481,-178.814,9.581,149.564
C09644=1113.021,218.136,-68.455,-178.816,9.578,149.564
C09645=1113.025,217.888,-68.429,-178.819,9.574,149.564
C09646=1113.030,217.638,-68.402,-178.821,9.571,149.564
C09647=1113.034,217.390,-68.376,-178.823,9.568,149.564
C09648=1113.038,217.141,-68.349,-178.825,9.566,149.564
C09649=1113.042,216.893,-68.323,-178.828,9.562,149.564
C09650=1113.047,216.644,-68.297,-178.830,9.559,149.564
C09651=1113.051,216.396,-68.270,-178.832,9.556,149.564
C09652=1113.056,216.147,-68.244,-178.834,9.554,149.564
C09653=1113.060,215.898,-68.219,-178.837,9.550,149.563
C09654=1113.064,215.650,-68.192,-178.839,9.547,149.563
C09655=1113.069,215.401,-68.166,-178.841,9.545,149.563
C09656=1113.073,215.153,-68.140,-178.843,9.541,149.563
C09657=1113.077,214.940,-68.117,-178.845,9.539,149.563
C09658=1113.080,214.726,-68.095,-178.847,9.536,149.563
C09659=1113.084,214.514,-68.073,-178.848,9.534,149.563
C09660=1113.088,214.300,-68.050,-178.850,9.532,149.563
C09661=1113.092,214.087,-68.028,-178.852,9.529,149.563
C09662=1113.096,213.874,-68.005,-178.854,9.526,149.562
C09663=1113.100,213.660,-67.983,-178.856,9.524,149.562
C09664=1113.103,213.447,-67.961,-178.858,9.521,149.562
C09665=1113.108,213.199,-67.934,-178.861,9.518,149.562
C09666=1113.112,212.951,-67.909,-178.863,9.515,149.562
C09667=1113.117,212.702,-67.883,-178.866,9.512,149.562
C09668=1113.121,212.453,-67.857,-178.869,9.509,149.562
C09669=1113.126,212.204,-67.830,-178.872,9.505,149.562
C09670=1113.130,211.956,-67.804,-178.875,9.503,149.562
C09671=1113.135,211.707,-67.779,-178.877,9.499,149.562
C09672=1113.139,211.459,-67.753,-178.880,9.497,149.562
C09673=1113.143,211.210,-67.727,-178.883,9.494,149.562
C09674=1113.147,210.961,-67.702,-178.885,9.491,149.562
C09675=1113.152,210.713,-67.675,-178.889,9.487,149.562
C09676=1113.157,210.464,-67.649,-178.891,9.484,149.562
C09677=1113.161,210.216,-67.623,-178.894,9.481,149.562
C09678=1113.165,209.967,-67.598,-178.897,9.478,149.563
C09679=1113.169,209.718,-67.572,-178.900,9.475,149.563
C09680=1113.174,209.469,-67.546,-178.903,9.473,149.563
C09681=1113.178,209.221,-67.521,-178.905,9.469,149.563
C09682=1113.183,208.972,-67.495,-178.908,9.467,149.563
C09683=1113.188,208.723,-67.469,-178.911,9.464,149.563
C09684=1113.193,208.475,-67.443,-178.914,9.461,149.563
C09685=1113.197,208.226,-67.418,-178.917,9.457,149.563
C09686=1113.201,207.978,-67.392,-178.920,9.455,149.563
C09687=1113.205,207.729,-67.366,-178.923,9.451,149.563
C09688=1113.210,207.481,-67.341,-178.926,9.449,149.563
C09689=1113.214,207.232,-67.315,-178.929,9.446,149.563
C09690=1113.218,206.983,-67.289,-178.931,9.443,149.563
C09691=1113.223,206.735,-67.264,-178.934,9.440,149.563
C09692=1113.228,206.486,-67.238,-178.937,9.437,149.564
C09693=1113.232,206.237,-67.212,-178.940,9.434,149.564
C09694=1113.237,205.989,-67.187,-178.943,9.432,149.564
C09695=1113.241,205.740,-67.162,-178.946,9.429,149.564
C09696=1113.245,205.491,-67.136,-178.948,9.426,149.564
C09697=1113.250,205.243,-67.111,-178.951,9.423,149.564
C09698=1113.254,204.994,-67.085,-178.954,9.420,149.564
C09699=1113.259,204.745,-67.059,-178.957,9.417,149.564
C09700=1113.263,204.497,-67.034,-178.960,9.415,149.564
C09701=1113.268,204.248,-67.009,-178.963,9.411,149.564
C09702=1113.272,203.999,-66.983,-178.966,9.408,149.564
C09703=1113.277,203.751,-66.958,-178.969,9.405,149.565
C09704=1113.280,203.502,-66.933,-178.972,9.403,149.565
C09705=1113.285,203.253,-66.908,-178.974,9.399,149.565
C09706=1113.290,203.005,-66.882,-178.977,9.397,149.565
C09707=1113.294,202.756,-66.856,-178.980,9.394,149.565
C09708=1113.299,202.507,-66.832,-178.983,9.391,149.565
C09709=1113.303,202.258,-66.806,-178.986,9.388,149.565
C09710=1113.308,202.010,-66.780,-178.989,9.385,149.565
C09711=1113.312,201.761,-66.756,-178.991,9.382,149.565
C09712=1113.316,201.512,-66.730,-178.994,9.380,149.565
C09713=1113.320,201.299,-66.709,-178.997,9.377,149.565
C09714=1113.324,201.086,-66.687,-178.999,9.374,149.565
C09715=1113.328,200.873,-66.666,-179.002,9.372,149.566
C09716=1113.332,200.660,-66.644,-179.004,9.369,149.565
C09717=1113.335,200.446,-66.623,-179.007,9.367,149.566
C09718=1113.339,200.233,-66.601,-179.009,9.364,149.566
C09719=1113.343,200.019,-66.579,-179.012,9.362,149.566
C09720=1113.347,199.806,-66.558,-179.014,9.358,149.566
C09721=1113.351,199.557,-66.533,-179.017,9.356,149.566
C09722=1113.357,199.309,-66.508,-179.020,9.353,149.566
C09723=1113.361,199.060,-66.482,-179.023,9.350,149.566
C09724=1113.365,198.811,-66.458,-179.025,9.347,149.566
C09725=1113.369,198.563,-66.432,-179.028,9.344,149.566
C09726=1113.375,198.314,-66.408,-179.031,9.341,149.566
C09727=1113.378,198.065,-66.382,-179.034,9.337,149.566
C09728=1113.383,197.817,-66.358,-179.037,9.334,149.566
C09729=1113.387,197.568,-66.332,-179.039,9.331,149.566
C09730=1113.392,197.319,-66.308,-179.042,9.328,149.566
C09731=1113.396,197.070,-66.283,-179.045,9.324,149.566
C09732=1113.401,196.822,-66.258,-179.048,9.321,149.566
C09733=1113.405,196.573,-66.233,-179.050,9.318,149.566
C09734=1113.410,196.324,-66.208,-179.053,9.315,149.566
C09735=1113.414,196.075,-66.183,-179.054,9.313,149.566
C09736=1113.419,195.827,-66.159,-179.057,9.309,149.566
C09737=1113.423,195.577,-66.134,-179.059,9.307,149.566
C09738=1113.427,195.330,-66.109,-179.061,9.304,149.565
C09739=1113.432,195.081,-66.084,-179.063,9.301,149.565
C09740=1113.437,194.832,-66.059,-179.065,9.298,149.565
C09741=1113.441,194.583,-66.035,-179.067,9.295,149.565
C09742=1113.446,194.334,-66.009,-179.069,9.293,149.565
C09743=1113.450,194.086,-65.985,-179.071,9.290,149.565
C09744=1113.455,193.836,-65.960,-179.073,9.288,149.565
C09745=1113.459,193.588,-65.936,-179.075,9.284,149.565
C09746=1113.464,193.340,-65.911,-179.077,9.282,149.565
C09747=1113.468,193.091,-65.886,-179.080,9.279,149.565
C09748=1113.473,192.842,-65.862,-179.082,9.276,149.564
C09749=1113.478,192.593,-65.837,-179.084,9.273,149.564
C09750=1113.482,192.344,-65.812,-179.086,9.271,149.564
C09751=1113.487,192.096,-65.788,-179.088,9.268,149.564
C09752=1113.490,191.847,-65.763,-179.090,9.265,149.564
C09753=1113.495,191.598,-65.738,-179.092,9.262,149.564
C09754=1113.500,191.350,-65.714,-179.094,9.260,149.564
C09755=1113.504,191.101,-65.689,-179.097,9.257,149.564
C09756=1113.509,190.852,-65.665,-179.099,9.254,149.564
C09757=1113.514,190.603,-65.640,-179.101,9.251,149.564
C09758=1113.518,190.354,-65.616,-179.103,9.249,149.564
C09759=1113.523,190.106,-65.591,-179.106,9.246,149.564
C09760=1113.527,189.857,-65.567,-179.108,9.243,149.564
C09761=1113.531,189.608,-65.542,-179.110,9.240,149.564
C09762=1113.536,189.359,-65.518,-179.113,9.237,149.564
C09763=1113.540,189.111,-65.494,-179.115,9.235,149.564
C09764=1113.545,188.861,-65.469,-179.117,9.232,149.564
C09765=1113.549,188.613,-65.445,-179.120,9.229,149.564
C09766=1113.554,188.364,-65.420,-179.121,9.226,149.563
C09767=1113.558,188.115,-65.396,-179.124,9.223,149.563
C09768=1113.563,187.867,-65.371,-179.126,9.221,149.563
C09769=1113.567,187.654,-65.350,-179.128,9.218,149.563
C09770=1113.571,187.440,-65.329,-179.130,9.215,149.563
C09771=1113.574,187.227,-65.308,-179.132,9.213,149.563
C09772=1113.578,187.013,-65.287,-179.134,9.211,149.563
C09773=1113.583,186.800,-65.267,-179.136,9.208,149.563
C09774=1113.586,186.587,-65.246,-179.138,9.206,149.563
C09775=1113.590,186.373,-65.225,-179.140,9.204,149.563
C09776=1113.594,186.159,-65.204,-179.142,9.201,149.563
C09777=1113.598,185.911,-65.180,-179.144,9.198,149.563
C09778=1113.603,185.663,-65.156,-179.147,9.195,149.563
C09779=1113.607,185.414,-65.132,-179.149,9.192,149.563
C09780=1113.612,185.164,-65.107,-179.151,9.190,149.563
C09781=1113.616,184.916,-65.083,-179.154,9.187,149.563
C09782=1113.621,184.667,-65.059,-179.157,9.184,149.563
C09783=1113.626,184.419,-65.034,-179.159,9.181,149.563
C09784=1113.630,184.169,-65.011,-179.162,9.178,149.563
C09785=1113.634,183.920,-64.987,-179.164,9.175,149.563
C09786=1113.639,183.672,-64.962,-179.166,9.172,149.563
C09787=1113.644,183.423,-64.938,-179.169,9.169,149.563
C09788=1113.649,183.174,-64.914,-179.171,9.166,149.563
C09789=1113.652,182.925,-64.890,-179.174,9.163,149.563
C09790=1113.657,182.677,-64.866,-179.176,9.161,149.563
C09791=1113.661,182.428,-64.843,-179.178,9.158,149.563
C09792=1113.667,182.179,-64.818,-179.181,9.154,149.563
C09793=1113.671,181.931,-64.794,-179.183,9.151,149.563
C09794=1113.676,181.682,-64.770,-179.186,9.148,149.563
C09795=1113.680,181.432,-64.746,-179.188,9.145,149.562
C09796=1113.684,181.184,-64.722,-179.191,9.142,149.562
C09797=1113.689,180.935,-64.699,-179.193,9.139,149.562
C09798=1113.694,180.686,-64.674,-179.196,9.136,149.562
C09799=1113.698,180.437,-64.651,-179.198,9.133,149.562
C09800=1113.703,180.189,-64.626,-179.201,9.130,149.562
C09801=1113.707,179.940,-64.602,-179.203,9.126,149.562
C09802=1113.711,179.691,-64.579,-179.206,9.123,149.562
C09803=1113.716,179.442,-64.555,-179.208,9.120,149.562
C09804=1113.720,179.193,-64.531,-179.210,9.117,149.562
C09805=1113.725,178.945,-64.507,-179.212,9.114,149.562
C09806=1113.730,178.696,-64.484,-179.215,9.111,149.562
C09807=1113.734,178.447,-64.460,-179.216,9.109,149.562
C09808=1113.739,178.198,-64.436,-179.219,9.105,149.562
C09809=1113.744,177.950,-64.412,-179.221,9.102,149.561
C09810=1113.748,177.700,-64.388,-179.223,9.100,149.561
C09811=1113.752,177.451,-64.364,-179.225,9.097,149.561
C09812=1113.757,177.202,-64.341,-179.228,9.093,149.561
C09813=1113.762,176.953,-64.317,-179.229,9.091,149.561
C09814=1113.766,176.705,-64.293,-179.232,9.088,149.561
C09815=1113.771,176.456,-64.270,-179.234,9.085,149.561
C09816=1113.775,176.208,-64.246,-179.236,9.082,149.561
C09817=1113.780,175.958,-64.222,-179.238,9.079,149.561
C09818=1113.785,175.709,-64.199,-179.241,9.076,149.561
C09819=1113.789,175.461,-64.175,-179.243,9.073,149.560
C09820=1113.794,175.212,-64.152,-179.245,9.070,149.560
C09821=1113.798,174.963,-64.128,-179.247,9.067,149.560
C09822=1113.802,174.715,-64.105,-179.249,9.064,149.560
C09823=1113.807,174.466,-64.081,-179.251,9.061,149.560
C09824=1113.811,174.217,-64.058,-179.254,9.058,149.560
C09825=1113.816,174.003,-64.038,-179.256,9.055,149.560
C09826=1113.819,173.790,-64.017,-179.257,9.053,149.560
C09827=1113.823,173.576,-63.997,-179.259,9.050,149.560
C09828=1113.828,173.363,-63.977,-179.261,9.048,149.560
C09829=1113.831,173.149,-63.957,-179.263,9.046,149.560
C09830=1113.835,172.936,-63.937,-179.264,9.043,149.559
C09831=1113.839,172.723,-63.917,-179.267,9.040,149.559
C09832=1113.843,172.509,-63.896,-179.269,9.038,149.559
C09833=1113.848,172.260,-63.873,-179.270,9.035,149.559
C09834=1113.852,172.011,-63.850,-179.273,9.032,149.559
C09835=1113.856,171.762,-63.826,-179.275,9.029,149.559
C09836=1113.861,171.513,-63.803,-179.278,9.026,149.559
C09837=1113.866,171.264,-63.779,-179.279,9.023,149.559
C09838=1113.870,171.015,-63.756,-179.282,9.020,149.559
C09839=1113.875,170.766,-63.733,-179.284,9.017,149.559
C09840=1113.879,170.518,-63.710,-179.286,9.014,149.558
C09841=1113.884,170.269,-63.687,-179.288,9.011,149.558
C09842=1113.888,170.020,-63.663,-179.291,9.008,149.558
C09843=1113.893,169.771,-63.640,-179.293,9.004,149.558
C09844=1113.897,169.522,-63.616,-179.295,9.002,149.558
C09845=1113.901,169.273,-63.593,-179.297,8.999,149.558
C09846=1113.906,169.024,-63.570,-179.299,8.995,149.558
C09847=1113.911,168.776,-63.547,-179.301,8.993,149.558
C09848=1113.916,168.527,-63.523,-179.304,8.990,149.558
C09849=1113.921,168.278,-63.500,-179.306,8.986,149.557
C09850=1113.925,168.029,-63.477,-179.308,8.983,149.557
C09851=1113.930,167.780,-63.454,-179.310,8.981,149.557
C09852=1113.934,167.531,-63.431,-179.312,8.977,149.557
C09853=1113.939,167.282,-63.407,-179.315,8.974,149.557
C09854=1113.943,167.033,-63.385,-179.317,8.971,149.557
C09855=1113.948,166.784,-63.362,-179.319,8.968,149.557
C09856=1113.953,166.535,-63.339,-179.321,8.965,149.557
C09857=1113.957,166.287,-63.316,-179.323,8.962,149.556
C09858=1113.962,166.038,-63.293,-179.326,8.959,149.556
C09859=1113.967,165.789,-63.269,-179.328,8.956,149.556
C09860=1113.970,165.540,-63.246,-179.330,8.953,149.556
C09861=1113.975,165.291,-63.223,-179.333,8.950,149.556
C09862=1113.980,165.043,-63.200,-179.335,8.946,149.556
C09863=1113.985,164.793,-63.178,-179.337,8.943,149.556
C09864=1113.989,164.544,-63.155,-179.339,8.941,149.556
C09865=1113.994,164.295,-63.131,-179.341,8.937,149.556
C09866=1113.998,164.046,-63.109,-179.344,8.934,149.556
C09867=1114.003,163.797,-63.085,-179.346,8.931,149.555
C09868=1114.008,163.549,-63.064,-179.348,8.928,149.555
C09869=1114.012,163.300,-63.040,-179.350,8.925,149.555
C09870=1114.017,163.051,-63.017,-179.352,8.922,149.555
C09871=1114.021,162.802,-62.994,-179.355,8.919,149.555
C09872=1114.026,162.552,-62.971,-179.357,8.915,149.555
C09873=1114.031,162.304,-62.949,-179.359,8.912,149.555
C09874=1114.035,162.055,-62.926,-179.361,8.909,149.554
C09875=1114.039,161.807,-62.903,-179.363,8.906,149.554
C09876=1114.044,161.557,-62.880,-179.365,8.903,149.554
C09877=1114.049,161.309,-62.858,-179.368,8.900,149.554
C09878=1114.054,161.060,-62.835,-179.370,8.896,149.554
C09879=1114.058,160.811,-62.812,-179.373,8.893,149.554
C09880=1114.063,160.561,-62.789,-179.375,8.890,149.554
C09881=1114.067,160.349,-62.770,-179.376,8.887,149.554
C09882=1114.071,160.134,-62.751,-179.378,8.885,149.553
C09883=1114.075,159.921,-62.731,-179.380,8.882,149.553
C09884=1114.079,159.707,-62.711,-179.382,8.879,149.553
C09885=1114.083,159.493,-62.692,-179.384,8.877,149.553
C09886=1114.086,159.281,-62.673,-179.386,8.873,149.553
C09887=1114.090,159.066,-62.654,-179.388,8.871,149.553
C09888=1114.094,158.853,-62.634,-179.390,8.868,149.553
C09889=1114.099,158.604,-62.611,-179.392,8.865,149.553
C09890=1114.104,158.355,-62.589,-179.394,8.862,149.553
C09891=1114.108,158.106,-62.566,-179.396,8.858,149.552
C09892=1114.113,157.857,-62.544,-179.398,8.855,149.552
C09893=1114.117,157.609,-62.521,-179.401,8.852,149.552
C09894=1114.122,157.359,-62.499,-179.403,8.848,149.552
C09895=1114.126,157.110,-62.476,-179.406,8.845,149.552
C09896=1114.132,156.861,-62.454,-179.408,8.842,149.551
C09897=1114.136,156.612,-62.432,-179.409,8.839,149.551
C09898=1114.140,156.363,-62.409,-179.412,8.836,149.551
C09899=1114.146,156.114,-62.387,-179.414,8.832,149.551
C09900=1114.150,155.866,-62.364,-179.416,8.829,149.551
C09901=1114.154,155.616,-62.342,-179.418,8.826,149.551
C09902=1114.159,155.367,-62.319,-179.420,8.822,149.550
C09903=1114.163,155.119,-62.297,-179.422,8.819,149.550
C09904=1114.168,154.869,-62.275,-179.425,8.816,149.550
C09905=1114.173,154.620,-62.252,-179.427,8.812,149.550
C09906=1114.177,154.372,-62.230,-179.429,8.809,149.550
C09907=1114.182,154.123,-62.208,-179.432,8.806,149.550
C09908=1114.186,153.874,-62.186,-179.434,8.802,149.549
C09909=1114.191,153.625,-62.163,-179.436,8.799,149.549
C09910=1114.196,153.376,-62.141,-179.438,8.795,149.549
C09911=1114.200,153.127,-62.119,-179.440,8.792,149.549
C09912=1114.206,152.878,-62.097,-179.443,8.788,149.549
C09913=1114.210,152.629,-62.074,-179.445,8.785,149.548
C09914=1114.215,152.380,-62.052,-179.447,8.782,149.548
C09915=1114.219,152.131,-62.030,-179.449,8.778,149.548
C09916=1114.224,151.881,-62.007,-179.451,8.775,149.548
C09917=1114.229,151.633,-61.985,-179.453,8.771,149.548
C09918=1114.233,151.384,-61.963,-179.455,8.768,149.548
C09919=1114.238,151.135,-61.941,-179.458,8.764,149.547
C09920=1114.242,150.886,-61.919,-179.460,8.760,149.547
C09921=1114.248,150.637,-61.897,-179.462,8.757,149.547
C09922=1114.252,150.388,-61.875,-179.465,8.754,149.547
C09923=1114.257,150.139,-61.853,-179.467,8.750,149.547
C09924=1114.261,149.890,-61.831,-179.469,8.747,149.546
C09925=1114.265,149.642,-61.809,-179.471,8.743,149.546
C09926=1114.270,149.392,-61.787,-179.473,8.740,149.546
C09927=1114.275,149.144,-61.765,-179.475,8.736,149.546
C09928=1114.280,148.894,-61.742,-179.477,8.733,149.545
C09929=1114.285,148.646,-61.721,-179.480,8.728,149.545
C09930=1114.289,148.396,-61.699,-179.482,8.725,149.545
C09931=1114.294,148.148,-61.677,-179.484,8.721,149.545
C09932=1114.298,147.898,-61.655,-179.486,8.718,149.544
C09933=1114.303,147.650,-61.633,-179.488,8.714,149.544
C09934=1114.307,147.400,-61.611,-179.490,8.711,149.544
C09935=1114.312,147.152,-61.589,-179.493,8.707,149.544
C09936=1114.317,146.903,-61.568,-179.495,8.703,149.543
C09937=1114.321,146.689,-61.549,-179.497,8.700,149.543
C09938=1114.324,146.475,-61.530,-179.499,8.697,149.543
C09939=1114.329,146.261,-61.512,-179.500,8.694,149.543
C09940=1114.332,146.048,-61.493,-179.502,8.691,149.543
C09941=1114.337,145.834,-61.474,-179.504,8.687,149.542
C09942=1114.341,145.620,-61.455,-179.506,8.685,149.542
C09943=1114.344,145.406,-61.437,-179.508,8.681,149.542
C09944=1114.349,145.193,-61.418,-179.509,8.678,149.542
C09945=1114.353,144.943,-61.396,-179.511,8.675,149.541
C09946=1114.358,144.695,-61.374,-179.513,8.671,149.541
C09947=1114.363,144.445,-61.353,-179.514,8.668,149.540
C09948=1114.368,144.196,-61.331,-179.516,8.664,149.540
C09949=1114.372,143.948,-61.310,-179.518,8.661,149.540
C09950=1114.377,143.699,-61.288,-179.519,8.658,149.540
C09951=1114.381,143.450,-61.266,-179.521,8.654,149.539
C09952=1114.386,143.200,-61.245,-179.523,8.651,149.539
C09953=1114.390,142.951,-61.223,-179.524,8.647,149.538
C09954=1114.395,142.702,-61.202,-179.526,8.644,149.538
C09955=1114.400,142.454,-61.180,-179.528,8.640,149.538
C09956=1114.405,142.204,-61.159,-179.529,8.637,149.538
C09957=1114.410,141.955,-61.137,-179.531,8.634,149.537
C09958=1114.414,141.707,-61.115,-179.533,8.630,149.537
C09959=1114.419,141.457,-61.094,-179.534,8.627,149.537
C09960=1114.423,141.208,-61.073,-179.536,8.623,149.536
C09961=1114.428,140.960,-61.051,-179.538,8.620,149.536
C09962=1114.432,140.710,-61.029,-179.539,8.617,149.536
C09963=1114.437,140.461,-61.008,-179.541,8.613,149.535
C09964=1114.442,140.212,-60.987,-179.542,8.610,149.535
C09965=1114.447,139.962,-60.965,-179.544,8.607,149.535
C09966=1114.451,139.714,-60.944,-179.546,8.603,149.534
C09967=1114.456,139.465,-60.922,-179.547,8.600,149.534
C09968=1114.460,139.215,-60.901,-179.549,8.597,149.534
C09969=1114.465,138.967,-60.879,-179.551,8.593,149.533
C09970=1114.470,138.718,-60.858,-179.552,8.590,149.533
C09971=1114.474,138.469,-60.837,-179.554,8.587,149.533
C09972=1114.479,138.220,-60.815,-179.556,8.583,149.532
C09973=1114.484,137.971,-60.794,-179.558,8.580,149.532
C09974=1114.489,137.722,-60.773,-179.560,8.577,149.532
C09975=1114.493,137.472,-60.752,-179.561,8.573,149.532
C09976=1114.498,137.224,-60.730,-179.563,8.570,149.531
C09977=1114.503,136.974,-60.709,-179.564,8.566,149.531
C09978=1114.508,136.726,-60.688,-179.566,8.563,149.531
C09979=1114.511,136.476,-60.667,-179.568,8.560,149.530
C09980=1114.516,136.227,-60.645,-179.570,8.556,149.530
C09981=1114.522,135.978,-60.624,-179.571,8.553,149.530
C09982=1114.526,135.730,-60.603,-179.573,8.550,149.530
C09983=1114.530,135.480,-60.582,-179.575,8.546,149.529
C09984=1114.535,135.231,-60.561,-179.576,8.543,149.529
C09985=1114.540,134.982,-60.539,-179.578,8.540,149.529
C09986=1114.545,134.733,-60.519,-179.580,8.536,149.528
C09987=1114.550,134.484,-60.497,-179.581,8.533,149.528
C09988=1114.554,134.234,-60.476,-179.583,8.530,149.528
C09989=1114.559,133.986,-60.455,-179.585,8.526,149.527
C09990=1114.563,133.737,-60.434,-179.586,8.523,149.527
C09991=1114.569,133.488,-60.413,-179.588,8.520,149.527
C09992=1114.573,133.239,-60.392,-179.591,8.516,149.527
C09993=1114.577,133.025,-60.373,-179.592,8.513,149.526
C09994=1114.581,132.811,-60.356,-179.593,8.510,149.526
C09995=1114.585,132.597,-60.337,-179.594,8.508,149.526
C09996=1114.589,132.383,-60.320,-179.596,8.505,149.525
//INST
///DATE 2021/06/15 17:29
///ATTR SC,RW,RJ
////FRAME ROBOT
///GROUP1 RB1
NOP
MOVL C00000 V=800.0 PL=0
MOVL C00001 V=800.0 PL=0
MOVL C00002 V=800.0 PL=0
MOVL C00003 V=800.0 PL=0
MOVL C00004 V=800.0 PL=0
MOVL C00005 V=800.0 PL=0
MOVL C00006 V=800.0 PL=0
MOVL C00007 V=800.0 PL=0
MOVL C00008 V=800.0 PL=0
MOVL C00009 V=800.0 PL=0
MOVL C00010 V=800.0 PL=0
MOVL C00011 V=800.0 PL=0
MOVL C00012 V=800.0 PL=0
MOVL C00013 V=800.0 PL=0
MOVL C00014 V=800.0 PL=0
MOVL C00015 V=800.0 PL=0
MOVL C00016 V=800.0 PL=0
MOVL C00017 V=800.0 PL=0
MOVL C00018 V=800.0 PL=0
MOVL C00019 V=800.0 PL=0
MOVL C00020 V=800.0 PL=0
MOVL C00021 V=800.0 PL=0
MOVL C00022 V=800.0 PL=0
MOVL C00023 V=800.0 PL=0
MOVL C00024 V=800.0 PL=0
MOVL C00025 V=800.0 PL=0
MOVL C00026 V=800.0 PL=0
MOVL C00027 V=800.0 PL=0
MOVL C00028 V=800.0 PL=0
MOVL C00029 V=800.0 PL=0
MOVL C00030 V=800.0 PL=0
MOVL C00031 V=800.0 PL=0
MOVL C00032 V=800.0 PL=0
MOVL C00033 V=800.0 PL=0
MOVL C00034 V=800.0 PL=0
MOVL C00035 V=800.0 PL=0
MOVL C00036 V=800.0 PL=0
MOVL C00037 V=800.0 PL=0
MOVL C00038 V=800.0 PL=0
MOVL C00039 V=800.0 PL=0
MOVL C00040 V=800.0 PL=0
MOVL C00041 V=800.0 PL=0
MOVL C00042 V=800.0 PL=0
MOVL C00043 V=800.0 PL=0
MOVL C00044 V=800.0 PL=0
MOVL C00045 V=800.0 PL=0
MOVL C00046 V=800.0 PL=0
MOVL C00047 V=800.0 PL=0
MOVL C00048 V=800.0 PL=0
MOVL C00049 V=800.0 PL=0
MOVL C00050 V=800.0 PL=0
MOVL C00051 V=800.0 PL=0
MOVL C00052 V=800.0 PL=0
MOVL C00053 V=800.0 PL=0
MOVL C00054 V=800.0 PL=0
MOVL C00055 V=800.0 PL=0
MOVL C00056 V=800.0 PL=0
MOVL C00057 V=800.0 PL=0
MOVL C00058 V=800.0 PL=0
MOVL C00059 V=800.0 PL=0
MOVL C00060 V=800.0 PL=0
MOVL C00061 V=800.0 PL=0
MOVL C00062 V=800.0 PL=0
MOVL C00063 V=800.0 PL=0
MOVL C00064 V=800.0 PL=0
MOVL C00065 V=800.0 PL=0
MOVL C00066 V=800.0 PL=0
MOVL C00067 V=800.0 PL=0
MOVL C00068 V=800.0 PL=0
MOVL C00069 V=800.0 PL=0
MOVL C00070 V=800.0 PL=0
MOVL C00071 V=800.0 PL=0
MOVL C00072 V=800.0 PL=0
MOVL C00073 V=800.0 PL=0
MOVL C00074 V=800.0 PL=0
MOVL C00075 V=800.0 PL=0
MOVL C00076 V=800.0 PL=0
MOVL C00077 V=800.0 PL=0
MOVL C00078 V=800.0 PL=0
MOVL C00079 V=800.0 PL=0
MOVL C00080 V=800.0 PL=0
MOVL C00081 V=800.0 PL=0
MOVL C00082 V=800.0 PL=0
MOVL C00083 V=800.0 PL=0
MOVL C00084 V=800.0 PL=0
MOVL C00085 V=800.0 PL=0
MOVL C00086 V=800.0 PL=0
MOVL C00087 V=800.0 PL=0
MOVL C00088 V=800.0 PL=0
MOVL C00089 V=800.0 PL=0
MOVL C00090 V=800.0 PL=0
MOVL C00091 V=800.0 PL=0
MOVL C00092 V=800.0 PL=0
MOVL C00093 V=800.0 PL=0
MOVL C00094 V=800.0 PL=0
MOVL C00095 V=800.0 PL=0
MOVL C00096 V=800.0 PL=0
MOVL C00097 V=800.0 PL=0
MOVL C00098 V=800.0 PL=0
MOVL C00099 V=800.0 PL=0
MOVL C00100 V=800.0 PL=0
MOVL C00101 V=800.0 PL=0
MOVL C00102 V=800.0 PL=0
MOVL C00103 V=800.0 PL=0
MOVL C00104 V=800.0 PL=0
MOVL C00105 V=800.0 PL=0
MOVL C00106 V=800.0 PL=0
MOVL C00107 V=800.0 PL=0
MOVL C00108 V=800.0 PL=0
MOVL C00109 V=800.0 PL=0
MOVL C00110 V=800.0 PL=0
MOVL C00111 V=800.0 PL=0
MOVL C00112 V=800.0 PL=0
MOVL C00113 V=800.0 PL=0
MOVL C00114 V=800.0 PL=0
MOVL C00115 V=800.0 PL=0
MOVL C00116 V=800.0 PL=0
MOVL C00117 V=800.0 PL=0
MOVL C00118 V=800.0 PL=0
MOVL C00119 V=800.0 PL=0
MOVL C00120 V=800.0 PL=0
MOVL C00121 V=800.0 PL=0
MOVL C00122 V=800.0 PL=0
MOVL C00123 V=800.0 PL=0
MOVL C00124 V=800.0 PL=0
MOVL C00125 V=800.0 PL=0
MOVL C00126 V=800.0 PL=0
MOVL C00127 V=800.0 PL=0
MOVL C00128 V=800.0 PL=0
MOVL C00129 V=800.0 PL=0
MOVL C00130 V=800.0 PL=0
MOVL C00131 V=800.0 PL=0
MOVL C00132 V=800.0 PL=0
MOVL C00133 V=800.0 PL=0
MOVL C00134 V=800.0 PL=0
MOVL C00135 V=800.0 PL=0
MOVL C00136 V=800.0 PL=0
MOVL C00137 V=800.0 PL=0
MOVL C00138 V=800.0 PL=0
MOVL C00139 V=800.0 PL=0
MOVL C00140 V=800.0 PL=0
MOVL C00141 V=800.0 PL=0
MOVL C00142 V=800.0 PL=0
MOVL C00143 V=800.0 PL=0
MOVL C00144 V=800.0 PL=0
MOVL C00145 V=800.0 PL=0
MOVL C00146 V=800.0 PL=0
MOVL C00147 V=800.0 PL=0
MOVL C00148 V=800.0 PL=0
MOVL C00149 V=800.0 PL=0
MOVL C00150 V=800.0 PL=0
MOVL C00151 V=800.0 PL=0
MOVL C00152 V=800.0 PL=0
MOVL C00153 V=800.0 PL=0
MOVL C00154 V=800.0 PL=0
MOVL C00155 V=800.0 PL=0
MOVL C00156 V=800.0 PL=0
MOVL C00157 V=800.0 PL=0
MOVL C00158 V=800.0 PL=0
MOVL C00159 V=800.0 PL=0
MOVL C00160 V=800.0 PL=0
MOVL C00161 V=800.0 PL=0
MOVL C00162 V=800.0 PL=0
MOVL C00163 V=800.0 PL=0
MOVL C00164 V=800.0 PL=0
MOVL C00165 V=800.0 PL=0
MOVL C00166 V=800.0 PL=0
MOVL C00167 V=800.0 PL=0
MOVL C00168 V=800.0 PL=0
MOVL C00169 V=800.0 PL=0
MOVL C00170 V=800.0 PL=0
MOVL C00171 V=800.0 PL=0
MOVL C00172 V=800.0 PL=0
MOVL C00173 V=800.0 PL=0
MOVL C00174 V=800.0 PL=0
MOVL C00175 V=800.0 PL=0
MOVL C00176 V=800.0 PL=0
MOVL C00177 V=800.0 PL=0
MOVL C00178 V=800.0 PL=0
MOVL C00179 V=800.0 PL=0
MOVL C00180 V=800.0 PL=0
MOVL C00181 V=800.0 PL=0
MOVL C00182 V=800.0 PL=0
MOVL C00183 V=800.0 PL=0
MOVL C00184 V=800.0 PL=0
MOVL C00185 V=800.0 PL=0
MOVL C00186 V=800.0 PL=0
MOVL C00187 V=800.0 PL=0
MOVL C00188 V=800.0 PL=0
MOVL C00189 V=800.0 PL=0
MOVL C00190 V=800.0 PL=0
MOVL C00191 V=800.0 PL=0
MOVL C00192 V=800.0 PL=0
MOVL C00193 V=800.0 PL=0
MOVL C00194 V=800.0 PL=0
MOVL C00195 V=800.0 PL=0
MOVL C00196 V=800.0 PL=0
MOVL C00197 V=800.0 PL=0
MOVL C00198 V=800.0 PL=0
MOVL C00199 V=800.0 PL=0
MOVL C00200 V=800.0 PL=0
MOVL C00201 V=800.0 PL=0
MOVL C00202 V=800.0 PL=0
MOVL C00203 V=800.0 PL=0
MOVL C00204 V=800.0 PL=0
MOVL C00205 V=800.0 PL=0
MOVL C00206 V=800.0 PL=0
MOVL C00207 V=800.0 PL=0
MOVL C00208 V=800.0 PL=0
MOVL C00209 V=800.0 PL=0
MOVL C00210 V=800.0 PL=0
MOVL C00211 V=800.0 PL=0
MOVL C00212 V=800.0 PL=0
MOVL C00213 V=800.0 PL=0
MOVL C00214 V=800.0 PL=0
MOVL C00215 V=800.0 PL=0
MOVL C00216 V=800.0 PL=0
MOVL C00217 V=800.0 PL=0
MOVL C00218 V=800.0 PL=0
MOVL C00219 V=800.0 PL=0
MOVL C00220 V=800.0 PL=0
MOVL C00221 V=800.0 PL=0
MOVL C00222 V=800.0 PL=0
MOVL C00223 V=800.0 PL=0
MOVL C00224 V=800.0 PL=0
MOVL C00225 V=800.0 PL=0
MOVL C00226 V=800.0 PL=0
MOVL C00227 V=800.0 PL=0
MOVL C00228 V=800.0 PL=0
MOVL C00229 V=800.0 PL=0
MOVL C00230 V=800.0 PL=0
MOVL C00231 V=800.0 PL=0
MOVL C00232 V=800.0 PL=0
MOVL C00233 V=800.0 PL=0
MOVL C00234 V=800.0 PL=0
MOVL C00235 V=800.0 PL=0
MOVL C00236 V=800.0 PL=0
MOVL C00237 V=800.0 PL=0
MOVL C00238 V=800.0 PL=0
MOVL C00239 V=800.0 PL=0
MOVL C00240 V=800.0 PL=0
MOVL C00241 V=800.0 PL=0
MOVL C00242 V=800.0 PL=0
MOVL C00243 V=800.0 PL=0
MOVL C00244 V=800.0 PL=0
MOVL C00245 V=800.0 PL=0
MOVL C00246 V=800.0 PL=0
MOVL C00247 V=800.0 PL=0
MOVL C00248 V=800.0 PL=0
MOVL C00249 V=800.0 PL=0
MOVL C00250 V=800.0 PL=0
MOVL C00251 V=800.0 PL=0
MOVL C00252 V=800.0 PL=0
MOVL C00253 V=800.0 PL=0
MOVL C00254 V=800.0 PL=0
MOVL C00255 V=800.0 PL=0
MOVL C00256 V=800.0 PL=0
MOVL C00257 V=800.0 PL=0
MOVL C00258 V=800.0 PL=0
MOVL C00259 V=800.0 PL=0
MOVL C00260 V=800.0 PL=0
MOVL C00261 V=800.0 PL=0
MOVL C00262 V=800.0 PL=0
MOVL C00263 V=800.0 PL=0
MOVL C00264 V=800.0 PL=0
MOVL C00265 V=800.0 PL=0
MOVL C00266 V=800.0 PL=0
MOVL C00267 V=800.0 PL=0
MOVL C00268 V=800.0 PL=0
MOVL C00269 V=800.0 PL=0
MOVL C00270 V=800.0 PL=0
MOVL C00271 V=800.0 PL=0
MOVL C00272 V=800.0 PL=0
MOVL C00273 V=800.0 PL=0
MOVL C00274 V=800.0 PL=0
MOVL C00275 V=800.0 PL=0
MOVL C00276 V=800.0 PL=0
MOVL C00277 V=800.0 PL=0
MOVL C00278 V=800.0 PL=0
MOVL C00279 V=800.0 PL=0
MOVL C00280 V=800.0 PL=0
MOVL C00281 V=800.0 PL=0
MOVL C00282 V=800.0 PL=0
MOVL C00283 V=800.0 PL=0
MOVL C00284 V=800.0 PL=0
MOVL C00285 V=800.0 PL=0
MOVL C00286 V=800.0 PL=0
MOVL C00287 V=800.0 PL=0
MOVL C00288 V=800.0 PL=0
MOVL C00289 V=800.0 PL=0
MOVL C00290 V=800.0 PL=0
MOVL C00291 V=800.0 PL=0
MOVL C00292 V=800.0 PL=0
MOVL C00293 V=800.0 PL=0
MOVL C00294 V=800.0 PL=0
MOVL C00295 V=800.0 PL=0
MOVL C00296 V=800.0 PL=0
MOVL C00297 V=800.0 PL=0
MOVL C00298 V=800.0 PL=0
MOVL C00299 V=800.0 PL=0
MOVL C00300 V=800.0 PL=0
MOVL C00301 V=800.0 PL=0
MOVL C00302 V=800.0 PL=0
MOVL C00303 V=800.0 PL=0
MOVL C00304 V=800.0 PL=0
MOVL C00305 V=800.0 PL=0
MOVL C00306 V=800.0 PL=0
MOVL C00307 V=800.0 PL=0
MOVL C00308 V=800.0 PL=0
MOVL C00309 V=800.0 PL=0
MOVL C00310 V=800.0 PL=0
MOVL C00311 V=800.0 PL=0
MOVL C00312 V=800.0 PL=0
MOVL C00313 V=800.0 PL=0
MOVL C00314 V=800.0 PL=0
MOVL C00315 V=800.0 PL=0
MOVL C00316 V=800.0 PL=0
MOVL C00317 V=800.0 PL=0
MOVL C00318 V=800.0 PL=0
MOVL C00319 V=800.0 PL=0
MOVL C00320 V=800.0 PL=0
MOVL C00321 V=800.0 PL=0
MOVL C00322 V=800.0 PL=0
MOVL C00323 V=800.0 PL=0
MOVL C00324 V=800.0 PL=0
MOVL C00325 V=800.0 PL=0
MOVL C00326 V=800.0 PL=0
MOVL C00327 V=800.0 PL=0
MOVL C00328 V=800.0 PL=0
MOVL C00329 V=800.0 PL=0
MOVL C00330 V=800.0 PL=0
MOVL C00331 V=800.0 PL=0
MOVL C00332 V=800.0 PL=0
MOVL C00333 V=800.0 PL=0
MOVL C00334 V=800.0 PL=0
MOVL C00335 V=800.0 PL=0
MOVL C00336 V=800.0 PL=0
MOVL C00337 V=800.0 PL=0
MOVL C00338 V=800.0 PL=0
MOVL C00339 V=800.0 PL=0
MOVL C00340 V=800.0 PL=0
MOVL C00341 V=800.0 PL=0
MOVL C00342 V=800.0 PL=0
MOVL C00343 V=800.0 PL=0
MOVL C00344 V=800.0 PL=0
MOVL C00345 V=800.0 PL=0
MOVL C00346 V=800.0 PL=0
MOVL C00347 V=800.0 PL=0
MOVL C00348 V=800.0 PL=0
MOVL C00349 V=800.0 PL=0
MOVL C00350 V=800.0 PL=0
MOVL C00351 V=800.0 PL=0
MOVL C00352 V=800.0 PL=0
MOVL C00353 V=800.0 PL=0
MOVL C00354 V=800.0 PL=0
MOVL C00355 V=800.0 PL=0
MOVL C00356 V=800.0 PL=0
MOVL C00357 V=800.0 PL=0
MOVL C00358 V=800.0 PL=0
MOVL C00359 V=800.0 PL=0
MOVL C00360 V=800.0 PL=0
MOVL C00361 V=800.0 PL=0
MOVL C00362 V=800.0 PL=0
MOVL C00363 V=800.0 PL=0
MOVL C00364 V=800.0 PL=0
MOVL C00365 V=800.0 PL=0
MOVL C00366 V=800.0 PL=0
MOVL C00367 V=800.0 PL=0
MOVL C00368 V=800.0 PL=0
MOVL C00369 V=800.0 PL=0
MOVL C00370 V=800.0 PL=0
MOVL C00371 V=800.0 PL=0
MOVL C00372 V=800.0 PL=0
MOVL C00373 V=800.0 PL=0
MOVL C00374 V=800.0 PL=0
MOVL C00375 V=800.0 PL=0
MOVL C00376 V=800.0 PL=0
MOVL C00377 V=800.0 PL=0
MOVL C00378 V=800.0 PL=0
MOVL C00379 V=800.0 PL=0
MOVL C00380 V=800.0 PL=0
MOVL C00381 V=800.0 PL=0
MOVL C00382 V=800.0 PL=0
MOVL C00383 V=800.0 PL=0
MOVL C00384 V=800.0 PL=0
MOVL C00385 V=800.0 PL=0
MOVL C00386 V=800.0 PL=0
MOVL C00387 V=800.0 PL=0
MOVL C00388 V=800.0 PL=0
MOVL C00389 V=800.0 PL=0
MOVL C00390 V=800.0 PL=0
MOVL C00391 V=800.0 PL=0
MOVL C00392 V=800.0 PL=0
MOVL C00393 V=800.0 PL=0
MOVL C00394 V=800.0 PL=0
MOVL C00395 V=800.0 PL=0
MOVL C00396 V=800.0 PL=0
MOVL C00397 V=800.0 PL=0
MOVL C00398 V=800.0 PL=0
MOVL C00399 V=800.0 PL=0
MOVL C00400 V=800.0 PL=0
MOVL C00401 V=800.0 PL=0
MOVL C00402 V=800.0 PL=0
MOVL C00403 V=800.0 PL=0
MOVL C00404 V=800.0 PL=0
MOVL C00405 V=800.0 PL=0
MOVL C00406 V=800.0 PL=0
MOVL C00407 V=800.0 PL=0
MOVL C00408 V=800.0 PL=0
MOVL C00409 V=800.0 PL=0
MOVL C00410 V=800.0 PL=0
MOVL C00411 V=800.0 PL=0
MOVL C00412 V=800.0 PL=0
MOVL C00413 V=800.0 PL=0
MOVL C00414 V=800.0 PL=0
MOVL C00415 V=800.0 PL=0
MOVL C00416 V=800.0 PL=0
MOVL C00417 V=800.0 PL=0
MOVL C00418 V=800.0 PL=0
MOVL C00419 V=800.0 PL=0
MOVL C00420 V=800.0 PL=0
MOVL C00421 V=800.0 PL=0
MOVL C00422 V=800.0 PL=0
MOVL C00423 V=800.0 PL=0
MOVL C00424 V=800.0 PL=0
MOVL C00425 V=800.0 PL=0
MOVL C00426 V=800.0 PL=0
MOVL C00427 V=800.0 PL=0
MOVL C00428 V=800.0 PL=0
MOVL C00429 V=800.0 PL=0
MOVL C00430 V=800.0 PL=0
MOVL C00431 V=800.0 PL=0
MOVL C00432 V=800.0 PL=0
MOVL C00433 V=800.0 PL=0
MOVL C00434 V=800.0 PL=0
MOVL C00435 V=800.0 PL=0
MOVL C00436 V=800.0 PL=0
MOVL C00437 V=800.0 PL=0
MOVL C00438 V=800.0 PL=0
MOVL C00439 V=800.0 PL=0
MOVL C00440 V=800.0 PL=0
MOVL C00441 V=800.0 PL=0
MOVL C00442 V=800.0 PL=0
MOVL C00443 V=800.0 PL=0
MOVL C00444 V=800.0 PL=0
MOVL C00445 V=800.0 PL=0
MOVL C00446 V=800.0 PL=0
MOVL C00447 V=800.0 PL=0
MOVL C00448 V=800.0 PL=0
MOVL C00449 V=800.0 PL=0
MOVL C00450 V=800.0 PL=0
MOVL C00451 V=800.0 PL=0
MOVL C00452 V=800.0 PL=0
MOVL C00453 V=800.0 PL=0
MOVL C00454 V=800.0 PL=0
MOVL C00455 V=800.0 PL=0
MOVL C00456 V=800.0 PL=0
MOVL C00457 V=800.0 PL=0
MOVL C00458 V=800.0 PL=0
MOVL C00459 V=800.0 PL=0
MOVL C00460 V=800.0 PL=0
MOVL C00461 V=800.0 PL=0
MOVL C00462 V=800.0 PL=0
MOVL C00463 V=800.0 PL=0
MOVL C00464 V=800.0 PL=0
MOVL C00465 V=800.0 PL=0
MOVL C00466 V=800.0 PL=0
MOVL C00467 V=800.0 PL=0
MOVL C00468 V=800.0 PL=0
MOVL C00469 V=800.0 PL=0
MOVL C00470 V=800.0 PL=0
MOVL C00471 V=800.0 PL=0
MOVL C00472 V=800.0 PL=0
MOVL C00473 V=800.0 PL=0
MOVL C00474 V=800.0 PL=0
MOVL C00475 V=800.0 PL=0
MOVL C00476 V=800.0 PL=0
MOVL C00477 V=800.0 PL=0
MOVL C00478 V=800.0 PL=0
MOVL C00479 V=800.0 PL=0
MOVL C00480 V=800.0 PL=0
MOVL C00481 V=800.0 PL=0
MOVL C00482 V=800.0 PL=0
MOVL C00483 V=800.0 PL=0
MOVL C00484 V=800.0 PL=0
MOVL C00485 V=800.0 PL=0
MOVL C00486 V=800.0 PL=0
MOVL C00487 V=800.0 PL=0
MOVL C00488 V=800.0 PL=0
MOVL C00489 V=800.0 PL=0
MOVL C00490 V=800.0 PL=0
MOVL C00491 V=800.0 PL=0
MOVL C00492 V=800.0 PL=0
MOVL C00493 V=800.0 PL=0
MOVL C00494 V=800.0 PL=0
MOVL C00495 V=800.0 PL=0
MOVL C00496 V=800.0 PL=0
MOVL C00497 V=800.0 PL=0
MOVL C00498 V=800.0 PL=0
MOVL C00499 V=800.0 PL=0
MOVL C00500 V=800.0 PL=0
MOVL C00501 V=800.0 PL=0
MOVL C00502 V=800.0 PL=0
MOVL C00503 V=800.0 PL=0
MOVL C00504 V=800.0 PL=0
MOVL C00505 V=800.0 PL=0
MOVL C00506 V=800.0 PL=0
MOVL C00507 V=800.0 PL=0
MOVL C00508 V=800.0 PL=0
MOVL C00509 V=800.0 PL=0
MOVL C00510 V=800.0 PL=0
MOVL C00511 V=800.0 PL=0
MOVL C00512 V=800.0 PL=0
MOVL C00513 V=800.0 PL=0
MOVL C00514 V=800.0 PL=0
MOVL C00515 V=800.0 PL=0
MOVL C00516 V=800.0 PL=0
MOVL C00517 V=800.0 PL=0
MOVL C00518 V=800.0 PL=0
MOVL C00519 V=800.0 PL=0
MOVL C00520 V=800.0 PL=0
MOVL C00521 V=800.0 PL=0
MOVL C00522 V=800.0 PL=0
MOVL C00523 V=800.0 PL=0
MOVL C00524 V=800.0 PL=0
MOVL C00525 V=800.0 PL=0
MOVL C00526 V=800.0 PL=0
MOVL C00527 V=800.0 PL=0
MOVL C00528 V=800.0 PL=0
MOVL C00529 V=800.0 PL=0
MOVL C00530 V=800.0 PL=0
MOVL C00531 V=800.0 PL=0
MOVL C00532 V=800.0 PL=0
MOVL C00533 V=800.0 PL=0
MOVL C00534 V=800.0 PL=0
MOVL C00535 V=800.0 PL=0
MOVL C00536 V=800.0 PL=0
MOVL C00537 V=800.0 PL=0
MOVL C00538 V=800.0 PL=0
MOVL C00539 V=800.0 PL=0
MOVL C00540 V=800.0 PL=0
MOVL C00541 V=800.0 PL=0
MOVL C00542 V=800.0 PL=0
MOVL C00543 V=800.0 PL=0
MOVL C00544 V=800.0 PL=0
MOVL C00545 V=800.0 PL=0
MOVL C00546 V=800.0 PL=0
MOVL C00547 V=800.0 PL=0
MOVL C00548 V=800.0 PL=0
MOVL C00549 V=800.0 PL=0
MOVL C00550 V=800.0 PL=0
MOVL C00551 V=800.0 PL=0
MOVL C00552 V=800.0 PL=0
MOVL C00553 V=800.0 PL=0
MOVL C00554 V=800.0 PL=0
MOVL C00555 V=800.0 PL=0
MOVL C00556 V=800.0 PL=0
MOVL C00557 V=800.0 PL=0
MOVL C00558 V=800.0 PL=0
MOVL C00559 V=800.0 PL=0
MOVL C00560 V=800.0 PL=0
MOVL C00561 V=800.0 PL=0
MOVL C00562 V=800.0 PL=0
MOVL C00563 V=800.0 PL=0
MOVL C00564 V=800.0 PL=0
MOVL C00565 V=800.0 PL=0
MOVL C00566 V=800.0 PL=0
MOVL C00567 V=800.0 PL=0
MOVL C00568 V=800.0 PL=0
MOVL C00569 V=800.0 PL=0
MOVL C00570 V=800.0 PL=0
MOVL C00571 V=800.0 PL=0
MOVL C00572 V=800.0 PL=0
MOVL C00573 V=800.0 PL=0
MOVL C00574 V=800.0 PL=0
MOVL C00575 V=800.0 PL=0
MOVL C00576 V=800.0 PL=0
MOVL C00577 V=800.0 PL=0
MOVL C00578 V=800.0 PL=0
MOVL C00579 V=800.0 PL=0
MOVL C00580 V=800.0 PL=0
MOVL C00581 V=800.0 PL=0
MOVL C00582 V=800.0 PL=0
MOVL C00583 V=800.0 PL=0
MOVL C00584 V=800.0 PL=0
MOVL C00585 V=800.0 PL=0
MOVL C00586 V=800.0 PL=0
MOVL C00587 V=800.0 PL=0
MOVL C00588 V=800.0 PL=0
MOVL C00589 V=800.0 PL=0
MOVL C00590 V=800.0 PL=0
MOVL C00591 V=800.0 PL=0
MOVL C00592 V=800.0 PL=0
MOVL C00593 V=800.0 PL=0
MOVL C00594 V=800.0 PL=0
MOVL C00595 V=800.0 PL=0
MOVL C00596 V=800.0 PL=0
MOVL C00597 V=800.0 PL=0
MOVL C00598 V=800.0 PL=0
MOVL C00599 V=800.0 PL=0
MOVL C00600 V=800.0 PL=0
MOVL C00601 V=800.0 PL=0
MOVL C00602 V=800.0 PL=0
MOVL C00603 V=800.0 PL=0
MOVL C00604 V=800.0 PL=0
MOVL C00605 V=800.0 PL=0
MOVL C00606 V=800.0 PL=0
MOVL C00607 V=800.0 PL=0
MOVL C00608 V=800.0 PL=0
MOVL C00609 V=800.0 PL=0
MOVL C00610 V=800.0 PL=0
MOVL C00611 V=800.0 PL=0
MOVL C00612 V=800.0 PL=0
MOVL C00613 V=800.0 PL=0
MOVL C00614 V=800.0 PL=0
MOVL C00615 V=800.0 PL=0
MOVL C00616 V=800.0 PL=0
MOVL C00617 V=800.0 PL=0
MOVL C00618 V=800.0 PL=0
MOVL C00619 V=800.0 PL=0
MOVL C00620 V=800.0 PL=0
MOVL C00621 V=800.0 PL=0
MOVL C00622 V=800.0 PL=0
MOVL C00623 V=800.0 PL=0
MOVL C00624 V=800.0 PL=0
MOVL C00625 V=800.0 PL=0
MOVL C00626 V=800.0 PL=0
MOVL C00627 V=800.0 PL=0
MOVL C00628 V=800.0 PL=0
MOVL C00629 V=800.0 PL=0
MOVL C00630 V=800.0 PL=0
MOVL C00631 V=800.0 PL=0
MOVL C00632 V=800.0 PL=0
MOVL C00633 V=800.0 PL=0
MOVL C00634 V=800.0 PL=0
MOVL C00635 V=800.0 PL=0
MOVL C00636 V=800.0 PL=0
MOVL C00637 V=800.0 PL=0
MOVL C00638 V=800.0 PL=0
MOVL C00639 V=800.0 PL=0
MOVL C00640 V=800.0 PL=0
MOVL C00641 V=800.0 PL=0
MOVL C00642 V=800.0 PL=0
MOVL C00643 V=800.0 PL=0
MOVL C00644 V=800.0 PL=0
MOVL C00645 V=800.0 PL=0
MOVL C00646 V=800.0 PL=0
MOVL C00647 V=800.0 PL=0
MOVL C00648 V=800.0 PL=0
MOVL C00649 V=800.0 PL=0
MOVL C00650 V=800.0 PL=0
MOVL C00651 V=800.0 PL=0
MOVL C00652 V=800.0 PL=0
MOVL C00653 V=800.0 PL=0
MOVL C00654 V=800.0 PL=0
MOVL C00655 V=800.0 PL=0
MOVL C00656 V=800.0 PL=0
MOVL C00657 V=800.0 PL=0
MOVL C00658 V=800.0 PL=0
MOVL C00659 V=800.0 PL=0
MOVL C00660 V=800.0 PL=0
MOVL C00661 V=800.0 PL=0
MOVL C00662 V=800.0 PL=0
MOVL C00663 V=800.0 PL=0
MOVL C00664 V=800.0 PL=0
MOVL C00665 V=800.0 PL=0
MOVL C00666 V=800.0 PL=0
MOVL C00667 V=800.0 PL=0
MOVL C00668 V=800.0 PL=0
MOVL C00669 V=800.0 PL=0
MOVL C00670 V=800.0 PL=0
MOVL C00671 V=800.0 PL=0
MOVL C00672 V=800.0 PL=0
MOVL C00673 V=800.0 PL=0
MOVL C00674 V=800.0 PL=0
MOVL C00675 V=800.0 PL=0
MOVL C00676 V=800.0 PL=0
MOVL C00677 V=800.0 PL=0
MOVL C00678 V=800.0 PL=0
MOVL C00679 V=800.0 PL=0
MOVL C00680 V=800.0 PL=0
MOVL C00681 V=800.0 PL=0
MOVL C00682 V=800.0 PL=0
MOVL C00683 V=800.0 PL=0
MOVL C00684 V=800.0 PL=0
MOVL C00685 V=800.0 PL=0
MOVL C00686 V=800.0 PL=0
MOVL C00687 V=800.0 PL=0
MOVL C00688 V=800.0 PL=0
MOVL C00689 V=800.0 PL=0
MOVL C00690 V=800.0 PL=0
MOVL C00691 V=800.0 PL=0
MOVL C00692 V=800.0 PL=0
MOVL C00693 V=800.0 PL=0
MOVL C00694 V=800.0 PL=0
MOVL C00695 V=800.0 PL=0
MOVL C00696 V=800.0 PL=0
MOVL C00697 V=800.0 PL=0
MOVL C00698 V=800.0 PL=0
MOVL C00699 V=800.0 PL=0
MOVL C00700 V=800.0 PL=0
MOVL C00701 V=800.0 PL=0
MOVL C00702 V=800.0 PL=0
MOVL C00703 V=800.0 PL=0
MOVL C00704 V=800.0 PL=0
MOVL C00705 V=800.0 PL=0
MOVL C00706 V=800.0 PL=0
MOVL C00707 V=800.0 PL=0
MOVL C00708 V=800.0 PL=0
MOVL C00709 V=800.0 PL=0
MOVL C00710 V=800.0 PL=0
MOVL C00711 V=800.0 PL=0
MOVL C00712 V=800.0 PL=0
MOVL C00713 V=800.0 PL=0
MOVL C00714 V=800.0 PL=0
MOVL C00715 V=800.0 PL=0
MOVL C00716 V=800.0 PL=0
MOVL C00717 V=800.0 PL=0
MOVL C00718 V=800.0 PL=0
MOVL C00719 V=800.0 PL=0
MOVL C00720 V=800.0 PL=0
MOVL C00721 V=800.0 PL=0
MOVL C00722 V=800.0 PL=0
MOVL C00723 V=800.0 PL=0
MOVL C00724 V=800.0 PL=0
MOVL C00725 V=800.0 PL=0
MOVL C00726 V=800.0 PL=0
MOVL C00727 V=800.0 PL=0
MOVL C00728 V=800.0 PL=0
MOVL C00729 V=800.0 PL=0
MOVL C00730 V=800.0 PL=0
MOVL C00731 V=800.0 PL=0
MOVL C00732 V=800.0 PL=0
MOVL C00733 V=800.0 PL=0
MOVL C00734 V=800.0 PL=0
MOVL C00735 V=800.0 PL=0
MOVL C00736 V=800.0 PL=0
MOVL C00737 V=800.0 PL=0
MOVL C00738 V=800.0 PL=0
MOVL C00739 V=800.0 PL=0
MOVL C00740 V=800.0 PL=0
MOVL C00741 V=800.0 PL=0
MOVL C00742 V=800.0 PL=0
MOVL C00743 V=800.0 PL=0
MOVL C00744 V=800.0 PL=0
MOVL C00745 V=800.0 PL=0
MOVL C00746 V=800.0 PL=0
MOVL C00747 V=800.0 PL=0
MOVL C00748 V=800.0 PL=0
MOVL C00749 V=800.0 PL=0
MOVL C00750 V=800.0 PL=0
MOVL C00751 V=800.0 PL=0
MOVL C00752 V=800.0 PL=0
MOVL C00753 V=800.0 PL=0
MOVL C00754 V=800.0 PL=0
MOVL C00755 V=800.0 PL=0
MOVL C00756 V=800.0 PL=0
MOVL C00757 V=800.0 PL=0
MOVL C00758 V=800.0 PL=0
MOVL C00759 V=800.0 PL=0
MOVL C00760 V=800.0 PL=0
MOVL C00761 V=800.0 PL=0
MOVL C00762 V=800.0 PL=0
MOVL C00763 V=800.0 PL=0
MOVL C00764 V=800.0 PL=0
MOVL C00765 V=800.0 PL=0
MOVL C00766 V=800.0 PL=0
MOVL C00767 V=800.0 PL=0
MOVL C00768 V=800.0 PL=0
MOVL C00769 V=800.0 PL=0
MOVL C00770 V=800.0 PL=0
MOVL C00771 V=800.0 PL=0
MOVL C00772 V=800.0 PL=0
MOVL C00773 V=800.0 PL=0
MOVL C00774 V=800.0 PL=0
MOVL C00775 V=800.0 PL=0
MOVL C00776 V=800.0 PL=0
MOVL C00777 V=800.0 PL=0
MOVL C00778 V=800.0 PL=0
MOVL C00779 V=800.0 PL=0
MOVL C00780 V=800.0 PL=0
MOVL C00781 V=800.0 PL=0
MOVL C00782 V=800.0 PL=0
MOVL C00783 V=800.0 PL=0
MOVL C00784 V=800.0 PL=0
MOVL C00785 V=800.0 PL=0
MOVL C00786 V=800.0 PL=0
MOVL C00787 V=800.0 PL=0
MOVL C00788 V=800.0 PL=0
MOVL C00789 V=800.0 PL=0
MOVL C00790 V=800.0 PL=0
MOVL C00791 V=800.0 PL=0
MOVL C00792 V=800.0 PL=0
MOVL C00793 V=800.0 PL=0
MOVL C00794 V=800.0 PL=0
MOVL C00795 V=800.0 PL=0
MOVL C00796 V=800.0 PL=0
MOVL C00797 V=800.0 PL=0
MOVL C00798 V=800.0 PL=0
MOVL C00799 V=800.0 PL=0
MOVL C00800 V=800.0 PL=0
MOVL C00801 V=800.0 PL=0
MOVL C00802 V=800.0 PL=0
MOVL C00803 V=800.0 PL=0
MOVL C00804 V=800.0 PL=0
MOVL C00805 V=800.0 PL=0
MOVL C00806 V=800.0 PL=0
MOVL C00807 V=800.0 PL=0
MOVL C00808 V=800.0 PL=0
MOVL C00809 V=800.0 PL=0
MOVL C00810 V=800.0 PL=0
MOVL C00811 V=800.0 PL=0
MOVL C00812 V=800.0 PL=0
MOVL C00813 V=800.0 PL=0
MOVL C00814 V=800.0 PL=0
MOVL C00815 V=800.0 PL=0
MOVL C00816 V=800.0 PL=0
MOVL C00817 V=800.0 PL=0
MOVL C00818 V=800.0 PL=0
MOVL C00819 V=800.0 PL=0
MOVL C00820 V=800.0 PL=0
MOVL C00821 V=800.0 PL=0
MOVL C00822 V=800.0 PL=0
MOVL C00823 V=800.0 PL=0
MOVL C00824 V=800.0 PL=0
MOVL C00825 V=800.0 PL=0
MOVL C00826 V=800.0 PL=0
MOVL C00827 V=800.0 PL=0
MOVL C00828 V=800.0 PL=0
MOVL C00829 V=800.0 PL=0
MOVL C00830 V=800.0 PL=0
MOVL C00831 V=800.0 PL=0
MOVL C00832 V=800.0 PL=0
MOVL C00833 V=800.0 PL=0
MOVL C00834 V=800.0 PL=0
MOVL C00835 V=800.0 PL=0
MOVL C00836 V=800.0 PL=0
MOVL C00837 V=800.0 PL=0
MOVL C00838 V=800.0 PL=0
MOVL C00839 V=800.0 PL=0
MOVL C00840 V=800.0 PL=0
MOVL C00841 V=800.0 PL=0
MOVL C00842 V=800.0 PL=0
MOVL C00843 V=800.0 PL=0
MOVL C00844 V=800.0 PL=0
MOVL C00845 V=800.0 PL=0
MOVL C00846 V=800.0 PL=0
MOVL C00847 V=800.0 PL=0
MOVL C00848 V=800.0 PL=0
MOVL C00849 V=800.0 PL=0
MOVL C00850 V=800.0 PL=0
MOVL C00851 V=800.0 PL=0
MOVL C00852 V=800.0 PL=0
MOVL C00853 V=800.0 PL=0
MOVL C00854 V=800.0 PL=0
MOVL C00855 V=800.0 PL=0
MOVL C00856 V=800.0 PL=0
MOVL C00857 V=800.0 PL=0
MOVL C00858 V=800.0 PL=0
MOVL C00859 V=800.0 PL=0
MOVL C00860 V=800.0 PL=0
MOVL C00861 V=800.0 PL=0
MOVL C00862 V=800.0 PL=0
MOVL C00863 V=800.0 PL=0
MOVL C00864 V=800.0 PL=0
MOVL C00865 V=800.0 PL=0
MOVL C00866 V=800.0 PL=0
MOVL C00867 V=800.0 PL=0
MOVL C00868 V=800.0 PL=0
MOVL C00869 V=800.0 PL=0
MOVL C00870 V=800.0 PL=0
MOVL C00871 V=800.0 PL=0
MOVL C00872 V=800.0 PL=0
MOVL C00873 V=800.0 PL=0
MOVL C00874 V=800.0 PL=0
MOVL C00875 V=800.0 PL=0
MOVL C00876 V=800.0 PL=0
MOVL C00877 V=800.0 PL=0
MOVL C00878 V=800.0 PL=0
MOVL C00879 V=800.0 PL=0
MOVL C00880 V=800.0 PL=0
MOVL C00881 V=800.0 PL=0
MOVL C00882 V=800.0 PL=0
MOVL C00883 V=800.0 PL=0
MOVL C00884 V=800.0 PL=0
MOVL C00885 V=800.0 PL=0
MOVL C00886 V=800.0 PL=0
MOVL C00887 V=800.0 PL=0
MOVL C00888 V=800.0 PL=0
MOVL C00889 V=800.0 PL=0
MOVL C00890 V=800.0 PL=0
MOVL C00891 V=800.0 PL=0
MOVL C00892 V=800.0 PL=0
MOVL C00893 V=800.0 PL=0
MOVL C00894 V=800.0 PL=0
MOVL C00895 V=800.0 PL=0
MOVL C00896 V=800.0 PL=0
MOVL C00897 V=800.0 PL=0
MOVL C00898 V=800.0 PL=0
MOVL C00899 V=800.0 PL=0
MOVL C00900 V=800.0 PL=0
MOVL C00901 V=800.0 PL=0
MOVL C00902 V=800.0 PL=0
MOVL C00903 V=800.0 PL=0
MOVL C00904 V=800.0 PL=0
MOVL C00905 V=800.0 PL=0
MOVL C00906 V=800.0 PL=0
MOVL C00907 V=800.0 PL=0
MOVL C00908 V=800.0 PL=0
MOVL C00909 V=800.0 PL=0
MOVL C00910 V=800.0 PL=0
MOVL C00911 V=800.0 PL=0
MOVL C00912 V=800.0 PL=0
MOVL C00913 V=800.0 PL=0
MOVL C00914 V=800.0 PL=0
MOVL C00915 V=800.0 PL=0
MOVL C00916 V=800.0 PL=0
MOVL C00917 V=800.0 PL=0
MOVL C00918 V=800.0 PL=0
MOVL C00919 V=800.0 PL=0
MOVL C00920 V=800.0 PL=0
MOVL C00921 V=800.0 PL=0
MOVL C00922 V=800.0 PL=0
MOVL C00923 V=800.0 PL=0
MOVL C00924 V=800.0 PL=0
MOVL C00925 V=800.0 PL=0
MOVL C00926 V=800.0 PL=0
MOVL C00927 V=800.0 PL=0
MOVL C00928 V=800.0 PL=0
MOVL C00929 V=800.0 PL=0
MOVL C00930 V=800.0 PL=0
MOVL C00931 V=800.0 PL=0
MOVL C00932 V=800.0 PL=0
MOVL C00933 V=800.0 PL=0
MOVL C00934 V=800.0 PL=0
MOVL C00935 V=800.0 PL=0
MOVL C00936 V=800.0 PL=0
MOVL C00937 V=800.0 PL=0
MOVL C00938 V=800.0 PL=0
MOVL C00939 V=800.0 PL=0
MOVL C00940 V=800.0 PL=0
MOVL C00941 V=800.0 PL=0
MOVL C00942 V=800.0 PL=0
MOVL C00943 V=800.0 PL=0
MOVL C00944 V=800.0 PL=0
MOVL C00945 V=800.0 PL=0
MOVL C00946 V=800.0 PL=0
MOVL C00947 V=800.0 PL=0
MOVL C00948 V=800.0 PL=0
MOVL C00949 V=800.0 PL=0
MOVL C00950 V=800.0 PL=0
MOVL C00951 V=800.0 PL=0
MOVL C00952 V=800.0 PL=0
MOVL C00953 V=800.0 PL=0
MOVL C00954 V=800.0 PL=0
MOVL C00955 V=800.0 PL=0
MOVL C00956 V=800.0 PL=0
MOVL C00957 V=800.0 PL=0
MOVL C00958 V=800.0 PL=0
MOVL C00959 V=800.0 PL=0
MOVL C00960 V=800.0 PL=0
MOVL C00961 V=800.0 PL=0
MOVL C00962 V=800.0 PL=0
MOVL C00963 V=800.0 PL=0
MOVL C00964 V=800.0 PL=0
MOVL C00965 V=800.0 PL=0
MOVL C00966 V=800.0 PL=0
MOVL C00967 V=800.0 PL=0
MOVL C00968 V=800.0 PL=0
MOVL C00969 V=800.0 PL=0
MOVL C00970 V=800.0 PL=0
MOVL C00971 V=800.0 PL=0
MOVL C00972 V=800.0 PL=0
MOVL C00973 V=800.0 PL=0
MOVL C00974 V=800.0 PL=0
MOVL C00975 V=800.0 PL=0
MOVL C00976 V=800.0 PL=0
MOVL C00977 V=800.0 PL=0
MOVL C00978 V=800.0 PL=0
MOVL C00979 V=800.0 PL=0
MOVL C00980 V=800.0 PL=0
MOVL C00981 V=800.0 PL=0
MOVL C00982 V=800.0 PL=0
MOVL C00983 V=800.0 PL=0
MOVL C00984 V=800.0 PL=0
MOVL C00985 V=800.0 PL=0
MOVL C00986 V=800.0 PL=0
MOVL C00987 V=800.0 PL=0
MOVL C00988 V=800.0 PL=0
MOVL C00989 V=800.0 PL=0
MOVL C00990 V=800.0 PL=0
MOVL C00991 V=800.0 PL=0
MOVL C00992 V=800.0 PL=0
MOVL C00993 V=800.0 PL=0
MOVL C00994 V=800.0 PL=0
MOVL C00995 V=800.0 PL=0
MOVL C00996 V=800.0 PL=0
MOVL C00997 V=800.0 PL=0
MOVL C00998 V=800.0 PL=0
MOVL C00999 V=800.0 PL=0
MOVL C01000 V=800.0 PL=0
MOVL C01001 V=800.0 PL=0
MOVL C01002 V=800.0 PL=0
MOVL C01003 V=800.0 PL=0
MOVL C01004 V=800.0 PL=0
MOVL C01005 V=800.0 PL=0
MOVL C01006 V=800.0 PL=0
MOVL C01007 V=800.0 PL=0
MOVL C01008 V=800.0 PL=0
MOVL C01009 V=800.0 PL=0
MOVL C01010 V=800.0 PL=0
MOVL C01011 V=800.0 PL=0
MOVL C01012 V=800.0 PL=0
MOVL C01013 V=800.0 PL=0
MOVL C01014 V=800.0 PL=0
MOVL C01015 V=800.0 PL=0
MOVL C01016 V=800.0 PL=0
MOVL C01017 V=800.0 PL=0
MOVL C01018 V=800.0 PL=0
MOVL C01019 V=800.0 PL=0
MOVL C01020 V=800.0 PL=0
MOVL C01021 V=800.0 PL=0
MOVL C01022 V=800.0 PL=0
MOVL C01023 V=800.0 PL=0
MOVL C01024 V=800.0 PL=0
MOVL C01025 V=800.0 PL=0
MOVL C01026 V=800.0 PL=0
MOVL C01027 V=800.0 PL=0
MOVL C01028 V=800.0 PL=0
MOVL C01029 V=800.0 PL=0
MOVL C01030 V=800.0 PL=0
MOVL C01031 V=800.0 PL=0
MOVL C01032 V=800.0 PL=0
MOVL C01033 V=800.0 PL=0
MOVL C01034 V=800.0 PL=0
MOVL C01035 V=800.0 PL=0
MOVL C01036 V=800.0 PL=0
MOVL C01037 V=800.0 PL=0
MOVL C01038 V=800.0 PL=0
MOVL C01039 V=800.0 PL=0
MOVL C01040 V=800.0 PL=0
MOVL C01041 V=800.0 PL=0
MOVL C01042 V=800.0 PL=0
MOVL C01043 V=800.0 PL=0
MOVL C01044 V=800.0 PL=0
MOVL C01045 V=800.0 PL=0
MOVL C01046 V=800.0 PL=0
MOVL C01047 V=800.0 PL=0
MOVL C01048 V=800.0 PL=0
MOVL C01049 V=800.0 PL=0
MOVL C01050 V=800.0 PL=0
MOVL C01051 V=800.0 PL=0
MOVL C01052 V=800.0 PL=0
MOVL C01053 V=800.0 PL=0
MOVL C01054 V=800.0 PL=0
MOVL C01055 V=800.0 PL=0
MOVL C01056 V=800.0 PL=0
MOVL C01057 V=800.0 PL=0
MOVL C01058 V=800.0 PL=0
MOVL C01059 V=800.0 PL=0
MOVL C01060 V=800.0 PL=0
MOVL C01061 V=800.0 PL=0
MOVL C01062 V=800.0 PL=0
MOVL C01063 V=800.0 PL=0
MOVL C01064 V=800.0 PL=0
MOVL C01065 V=800.0 PL=0
MOVL C01066 V=800.0 PL=0
MOVL C01067 V=800.0 PL=0
MOVL C01068 V=800.0 PL=0
MOVL C01069 V=800.0 PL=0
MOVL C01070 V=800.0 PL=0
MOVL C01071 V=800.0 PL=0
MOVL C01072 V=800.0 PL=0
MOVL C01073 V=800.0 PL=0
MOVL C01074 V=800.0 PL=0
MOVL C01075 V=800.0 PL=0
MOVL C01076 V=800.0 PL=0
MOVL C01077 V=800.0 PL=0
MOVL C01078 V=800.0 PL=0
MOVL C01079 V=800.0 PL=0
MOVL C01080 V=800.0 PL=0
MOVL C01081 V=800.0 PL=0
MOVL C01082 V=800.0 PL=0
MOVL C01083 V=800.0 PL=0
MOVL C01084 V=800.0 PL=0
MOVL C01085 V=800.0 PL=0
MOVL C01086 V=800.0 PL=0
MOVL C01087 V=800.0 PL=0
MOVL C01088 V=800.0 PL=0
MOVL C01089 V=800.0 PL=0
MOVL C01090 V=800.0 PL=0
MOVL C01091 V=800.0 PL=0
MOVL C01092 V=800.0 PL=0
MOVL C01093 V=800.0 PL=0
MOVL C01094 V=800.0 PL=0
MOVL C01095 V=800.0 PL=0
MOVL C01096 V=800.0 PL=0
MOVL C01097 V=800.0 PL=0
MOVL C01098 V=800.0 PL=0
MOVL C01099 V=800.0 PL=0
MOVL C01100 V=800.0 PL=0
MOVL C01101 V=800.0 PL=0
MOVL C01102 V=800.0 PL=0
MOVL C01103 V=800.0 PL=0
MOVL C01104 V=800.0 PL=0
MOVL C01105 V=800.0 PL=0
MOVL C01106 V=800.0 PL=0
MOVL C01107 V=800.0 PL=0
MOVL C01108 V=800.0 PL=0
MOVL C01109 V=800.0 PL=0
MOVL C01110 V=800.0 PL=0
MOVL C01111 V=800.0 PL=0
MOVL C01112 V=800.0 PL=0
MOVL C01113 V=800.0 PL=0
MOVL C01114 V=800.0 PL=0
MOVL C01115 V=800.0 PL=0
MOVL C01116 V=800.0 PL=0
MOVL C01117 V=800.0 PL=0
MOVL C01118 V=800.0 PL=0
MOVL C01119 V=800.0 PL=0
MOVL C01120 V=800.0 PL=0
MOVL C01121 V=800.0 PL=0
MOVL C01122 V=800.0 PL=0
MOVL C01123 V=800.0 PL=0
MOVL C01124 V=800.0 PL=0
MOVL C01125 V=800.0 PL=0
MOVL C01126 V=800.0 PL=0
MOVL C01127 V=800.0 PL=0
MOVL C01128 V=800.0 PL=0
MOVL C01129 V=800.0 PL=0
MOVL C01130 V=800.0 PL=0
MOVL C01131 V=800.0 PL=0
MOVL C01132 V=800.0 PL=0
MOVL C01133 V=800.0 PL=0
MOVL C01134 V=800.0 PL=0
MOVL C01135 V=800.0 PL=0
MOVL C01136 V=800.0 PL=0
MOVL C01137 V=800.0 PL=0
MOVL C01138 V=800.0 PL=0
MOVL C01139 V=800.0 PL=0
MOVL C01140 V=800.0 PL=0
MOVL C01141 V=800.0 PL=0
MOVL C01142 V=800.0 PL=0
MOVL C01143 V=800.0 PL=0
MOVL C01144 V=800.0 PL=0
MOVL C01145 V=800.0 PL=0
MOVL C01146 V=800.0 PL=0
MOVL C01147 V=800.0 PL=0
MOVL C01148 V=800.0 PL=0
MOVL C01149 V=800.0 PL=0
MOVL C01150 V=800.0 PL=0
MOVL C01151 V=800.0 PL=0
MOVL C01152 V=800.0 PL=0
MOVL C01153 V=800.0 PL=0
MOVL C01154 V=800.0 PL=0
MOVL C01155 V=800.0 PL=0
MOVL C01156 V=800.0 PL=0
MOVL C01157 V=800.0 PL=0
MOVL C01158 V=800.0 PL=0
MOVL C01159 V=800.0 PL=0
MOVL C01160 V=800.0 PL=0
MOVL C01161 V=800.0 PL=0
MOVL C01162 V=800.0 PL=0
MOVL C01163 V=800.0 PL=0
MOVL C01164 V=800.0 PL=0
MOVL C01165 V=800.0 PL=0
MOVL C01166 V=800.0 PL=0
MOVL C01167 V=800.0 PL=0
MOVL C01168 V=800.0 PL=0
MOVL C01169 V=800.0 PL=0
MOVL C01170 V=800.0 PL=0
MOVL C01171 V=800.0 PL=0
MOVL C01172 V=800.0 PL=0
MOVL C01173 V=800.0 PL=0
MOVL C01174 V=800.0 PL=0
MOVL C01175 V=800.0 PL=0
MOVL C01176 V=800.0 PL=0
MOVL C01177 V=800.0 PL=0
MOVL C01178 V=800.0 PL=0
MOVL C01179 V=800.0 PL=0
MOVL C01180 V=800.0 PL=0
MOVL C01181 V=800.0 PL=0
MOVL C01182 V=800.0 PL=0
MOVL C01183 V=800.0 PL=0
MOVL C01184 V=800.0 PL=0
MOVL C01185 V=800.0 PL=0
MOVL C01186 V=800.0 PL=0
MOVL C01187 V=800.0 PL=0
MOVL C01188 V=800.0 PL=0
MOVL C01189 V=800.0 PL=0
MOVL C01190 V=800.0 PL=0
MOVL C01191 V=800.0 PL=0
MOVL C01192 V=800.0 PL=0
MOVL C01193 V=800.0 PL=0
MOVL C01194 V=800.0 PL=0
MOVL C01195 V=800.0 PL=0
MOVL C01196 V=800.0 PL=0
MOVL C01197 V=800.0 PL=0
MOVL C01198 V=800.0 PL=0
MOVL C01199 V=800.0 PL=0
MOVL C01200 V=800.0 PL=0
MOVL C01201 V=800.0 PL=0
MOVL C01202 V=800.0 PL=0
MOVL C01203 V=800.0 PL=0
MOVL C01204 V=800.0 PL=0
MOVL C01205 V=800.0 PL=0
MOVL C01206 V=800.0 PL=0
MOVL C01207 V=800.0 PL=0
MOVL C01208 V=800.0 PL=0
MOVL C01209 V=800.0 PL=0
MOVL C01210 V=800.0 PL=0
MOVL C01211 V=800.0 PL=0
MOVL C01212 V=800.0 PL=0
MOVL C01213 V=800.0 PL=0
MOVL C01214 V=800.0 PL=0
MOVL C01215 V=800.0 PL=0
MOVL C01216 V=800.0 PL=0
MOVL C01217 V=800.0 PL=0
MOVL C01218 V=800.0 PL=0
MOVL C01219 V=800.0 PL=0
MOVL C01220 V=800.0 PL=0
MOVL C01221 V=800.0 PL=0
MOVL C01222 V=800.0 PL=0
MOVL C01223 V=800.0 PL=0
MOVL C01224 V=800.0 PL=0
MOVL C01225 V=800.0 PL=0
MOVL C01226 V=800.0 PL=0
MOVL C01227 V=800.0 PL=0
MOVL C01228 V=800.0 PL=0
MOVL C01229 V=800.0 PL=0
MOVL C01230 V=800.0 PL=0
MOVL C01231 V=800.0 PL=0
MOVL C01232 V=800.0 PL=0
MOVL C01233 V=800.0 PL=0
MOVL C01234 V=800.0 PL=0
MOVL C01235 V=800.0 PL=0
MOVL C01236 V=800.0 PL=0
MOVL C01237 V=800.0 PL=0
MOVL C01238 V=800.0 PL=0
MOVL C01239 V=800.0 PL=0
MOVL C01240 V=800.0 PL=0
MOVL C01241 V=800.0 PL=0
MOVL C01242 V=800.0 PL=0
MOVL C01243 V=800.0 PL=0
MOVL C01244 V=800.0 PL=0
MOVL C01245 V=800.0 PL=0
MOVL C01246 V=800.0 PL=0
MOVL C01247 V=800.0 PL=0
MOVL C01248 V=800.0 PL=0
MOVL C01249 V=800.0 PL=0
MOVL C01250 V=800.0 PL=0
MOVL C01251 V=800.0 PL=0
MOVL C01252 V=800.0 PL=0
MOVL C01253 V=800.0 PL=0
MOVL C01254 V=800.0 PL=0
MOVL C01255 V=800.0 PL=0
MOVL C01256 V=800.0 PL=0
MOVL C01257 V=800.0 PL=0
MOVL C01258 V=800.0 PL=0
MOVL C01259 V=800.0 PL=0
MOVL C01260 V=800.0 PL=0
MOVL C01261 V=800.0 PL=0
MOVL C01262 V=800.0 PL=0
MOVL C01263 V=800.0 PL=0
MOVL C01264 V=800.0 PL=0
MOVL C01265 V=800.0 PL=0
MOVL C01266 V=800.0 PL=0
MOVL C01267 V=800.0 PL=0
MOVL C01268 V=800.0 PL=0
MOVL C01269 V=800.0 PL=0
MOVL C01270 V=800.0 PL=0
MOVL C01271 V=800.0 PL=0
MOVL C01272 V=800.0 PL=0
MOVL C01273 V=800.0 PL=0
MOVL C01274 V=800.0 PL=0
MOVL C01275 V=800.0 PL=0
MOVL C01276 V=800.0 PL=0
MOVL C01277 V=800.0 PL=0
MOVL C01278 V=800.0 PL=0
MOVL C01279 V=800.0 PL=0
MOVL C01280 V=800.0 PL=0
MOVL C01281 V=800.0 PL=0
MOVL C01282 V=800.0 PL=0
MOVL C01283 V=800.0 PL=0
MOVL C01284 V=800.0 PL=0
MOVL C01285 V=800.0 PL=0
MOVL C01286 V=800.0 PL=0
MOVL C01287 V=800.0 PL=0
MOVL C01288 V=800.0 PL=0
MOVL C01289 V=800.0 PL=0
MOVL C01290 V=800.0 PL=0
MOVL C01291 V=800.0 PL=0
MOVL C01292 V=800.0 PL=0
MOVL C01293 V=800.0 PL=0
MOVL C01294 V=800.0 PL=0
MOVL C01295 V=800.0 PL=0
MOVL C01296 V=800.0 PL=0
MOVL C01297 V=800.0 PL=0
MOVL C01298 V=800.0 PL=0
MOVL C01299 V=800.0 PL=0
MOVL C01300 V=800.0 PL=0
MOVL C01301 V=800.0 PL=0
MOVL C01302 V=800.0 PL=0
MOVL C01303 V=800.0 PL=0
MOVL C01304 V=800.0 PL=0
MOVL C01305 V=800.0 PL=0
MOVL C01306 V=800.0 PL=0
MOVL C01307 V=800.0 PL=0
MOVL C01308 V=800.0 PL=0
MOVL C01309 V=800.0 PL=0
MOVL C01310 V=800.0 PL=0
MOVL C01311 V=800.0 PL=0
MOVL C01312 V=800.0 PL=0
MOVL C01313 V=800.0 PL=0
MOVL C01314 V=800.0 PL=0
MOVL C01315 V=800.0 PL=0
MOVL C01316 V=800.0 PL=0
MOVL C01317 V=800.0 PL=0
MOVL C01318 V=800.0 PL=0
MOVL C01319 V=800.0 PL=0
MOVL C01320 V=800.0 PL=0
MOVL C01321 V=800.0 PL=0
MOVL C01322 V=800.0 PL=0
MOVL C01323 V=800.0 PL=0
MOVL C01324 V=800.0 PL=0
MOVL C01325 V=800.0 PL=0
MOVL C01326 V=800.0 PL=0
MOVL C01327 V=800.0 PL=0
MOVL C01328 V=800.0 PL=0
MOVL C01329 V=800.0 PL=0
MOVL C01330 V=800.0 PL=0
MOVL C01331 V=800.0 PL=0
MOVL C01332 V=800.0 PL=0
MOVL C01333 V=800.0 PL=0
MOVL C01334 V=800.0 PL=0
MOVL C01335 V=800.0 PL=0
MOVL C01336 V=800.0 PL=0
MOVL C01337 V=800.0 PL=0
MOVL C01338 V=800.0 PL=0
MOVL C01339 V=800.0 PL=0
MOVL C01340 V=800.0 PL=0
MOVL C01341 V=800.0 PL=0
MOVL C01342 V=800.0 PL=0
MOVL C01343 V=800.0 PL=0
MOVL C01344 V=800.0 PL=0
MOVL C01345 V=800.0 PL=0
MOVL C01346 V=800.0 PL=0
MOVL C01347 V=800.0 PL=0
MOVL C01348 V=800.0 PL=0
MOVL C01349 V=800.0 PL=0
MOVL C01350 V=800.0 PL=0
MOVL C01351 V=800.0 PL=0
MOVL C01352 V=800.0 PL=0
MOVL C01353 V=800.0 PL=0
MOVL C01354 V=800.0 PL=0
MOVL C01355 V=800.0 PL=0
MOVL C01356 V=800.0 PL=0
MOVL C01357 V=800.0 PL=0
MOVL C01358 V=800.0 PL=0
MOVL C01359 V=800.0 PL=0
MOVL C01360 V=800.0 PL=0
MOVL C01361 V=800.0 PL=0
MOVL C01362 V=800.0 PL=0
MOVL C01363 V=800.0 PL=0
MOVL C01364 V=800.0 PL=0
MOVL C01365 V=800.0 PL=0
MOVL C01366 V=800.0 PL=0
MOVL C01367 V=800.0 PL=0
MOVL C01368 V=800.0 PL=0
MOVL C01369 V=800.0 PL=0
MOVL C01370 V=800.0 PL=0
MOVL C01371 V=800.0 PL=0
MOVL C01372 V=800.0 PL=0
MOVL C01373 V=800.0 PL=0
MOVL C01374 V=800.0 PL=0
MOVL C01375 V=800.0 PL=0
MOVL C01376 V=800.0 PL=0
MOVL C01377 V=800.0 PL=0
MOVL C01378 V=800.0 PL=0
MOVL C01379 V=800.0 PL=0
MOVL C01380 V=800.0 PL=0
MOVL C01381 V=800.0 PL=0
MOVL C01382 V=800.0 PL=0
MOVL C01383 V=800.0 PL=0
MOVL C01384 V=800.0 PL=0
MOVL C01385 V=800.0 PL=0
MOVL C01386 V=800.0 PL=0
MOVL C01387 V=800.0 PL=0
MOVL C01388 V=800.0 PL=0
MOVL C01389 V=800.0 PL=0
MOVL C01390 V=800.0 PL=0
MOVL C01391 V=800.0 PL=0
MOVL C01392 V=800.0 PL=0
MOVL C01393 V=800.0 PL=0
MOVL C01394 V=800.0 PL=0
MOVL C01395 V=800.0 PL=0
MOVL C01396 V=800.0 PL=0
MOVL C01397 V=800.0 PL=0
MOVL C01398 V=800.0 PL=0
MOVL C01399 V=800.0 PL=0
MOVL C01400 V=800.0 PL=0
MOVL C01401 V=800.0 PL=0
MOVL C01402 V=800.0 PL=0
MOVL C01403 V=800.0 PL=0
MOVL C01404 V=800.0 PL=0
MOVL C01405 V=800.0 PL=0
MOVL C01406 V=800.0 PL=0
MOVL C01407 V=800.0 PL=0
MOVL C01408 V=800.0 PL=0
MOVL C01409 V=800.0 PL=0
MOVL C01410 V=800.0 PL=0
MOVL C01411 V=800.0 PL=0
MOVL C01412 V=800.0 PL=0
MOVL C01413 V=800.0 PL=0
MOVL C01414 V=800.0 PL=0
MOVL C01415 V=800.0 PL=0
MOVL C01416 V=800.0 PL=0
MOVL C01417 V=800.0 PL=0
MOVL C01418 V=800.0 PL=0
MOVL C01419 V=800.0 PL=0
MOVL C01420 V=800.0 PL=0
MOVL C01421 V=800.0 PL=0
MOVL C01422 V=800.0 PL=0
MOVL C01423 V=800.0 PL=0
MOVL C01424 V=800.0 PL=0
MOVL C01425 V=800.0 PL=0
MOVL C01426 V=800.0 PL=0
MOVL C01427 V=800.0 PL=0
MOVL C01428 V=800.0 PL=0
MOVL C01429 V=800.0 PL=0
MOVL C01430 V=800.0 PL=0
MOVL C01431 V=800.0 PL=0
MOVL C01432 V=800.0 PL=0
MOVL C01433 V=800.0 PL=0
MOVL C01434 V=800.0 PL=0
MOVL C01435 V=800.0 PL=0
MOVL C01436 V=800.0 PL=0
MOVL C01437 V=800.0 PL=0
MOVL C01438 V=800.0 PL=0
MOVL C01439 V=800.0 PL=0
MOVL C01440 V=800.0 PL=0
MOVL C01441 V=800.0 PL=0
MOVL C01442 V=800.0 PL=0
MOVL C01443 V=800.0 PL=0
MOVL C01444 V=800.0 PL=0
MOVL C01445 V=800.0 PL=0
MOVL C01446 V=800.0 PL=0
MOVL C01447 V=800.0 PL=0
MOVL C01448 V=800.0 PL=0
MOVL C01449 V=800.0 PL=0
MOVL C01450 V=800.0 PL=0
MOVL C01451 V=800.0 PL=0
MOVL C01452 V=800.0 PL=0
MOVL C01453 V=800.0 PL=0
MOVL C01454 V=800.0 PL=0
MOVL C01455 V=800.0 PL=0
MOVL C01456 V=800.0 PL=0
MOVL C01457 V=800.0 PL=0
MOVL C01458 V=800.0 PL=0
MOVL C01459 V=800.0 PL=0
MOVL C01460 V=800.0 PL=0
MOVL C01461 V=800.0 PL=0
MOVL C01462 V=800.0 PL=0
MOVL C01463 V=800.0 PL=0
MOVL C01464 V=800.0 PL=0
MOVL C01465 V=800.0 PL=0
MOVL C01466 V=800.0 PL=0
MOVL C01467 V=800.0 PL=0
MOVL C01468 V=800.0 PL=0
MOVL C01469 V=800.0 PL=0
MOVL C01470 V=800.0 PL=0
MOVL C01471 V=800.0 PL=0
MOVL C01472 V=800.0 PL=0
MOVL C01473 V=800.0 PL=0
MOVL C01474 V=800.0 PL=0
MOVL C01475 V=800.0 PL=0
MOVL C01476 V=800.0 PL=0
MOVL C01477 V=800.0 PL=0
MOVL C01478 V=800.0 PL=0
MOVL C01479 V=800.0 PL=0
MOVL C01480 V=800.0 PL=0
MOVL C01481 V=800.0 PL=0
MOVL C01482 V=800.0 PL=0
MOVL C01483 V=800.0 PL=0
MOVL C01484 V=800.0 PL=0
MOVL C01485 V=800.0 PL=0
MOVL C01486 V=800.0 PL=0
MOVL C01487 V=800.0 PL=0
MOVL C01488 V=800.0 PL=0
MOVL C01489 V=800.0 PL=0
MOVL C01490 V=800.0 PL=0
MOVL C01491 V=800.0 PL=0
MOVL C01492 V=800.0 PL=0
MOVL C01493 V=800.0 PL=0
MOVL C01494 V=800.0 PL=0
MOVL C01495 V=800.0 PL=0
MOVL C01496 V=800.0 PL=0
MOVL C01497 V=800.0 PL=0
MOVL C01498 V=800.0 PL=0
MOVL C01499 V=800.0 PL=0
MOVL C01500 V=800.0 PL=0
MOVL C01501 V=800.0 PL=0
MOVL C01502 V=800.0 PL=0
MOVL C01503 V=800.0 PL=0
MOVL C01504 V=800.0 PL=0
MOVL C01505 V=800.0 PL=0
MOVL C01506 V=800.0 PL=0
MOVL C01507 V=800.0 PL=0
MOVL C01508 V=800.0 PL=0
MOVL C01509 V=800.0 PL=0
MOVL C01510 V=800.0 PL=0
MOVL C01511 V=800.0 PL=0
MOVL C01512 V=800.0 PL=0
MOVL C01513 V=800.0 PL=0
MOVL C01514 V=800.0 PL=0
MOVL C01515 V=800.0 PL=0
MOVL C01516 V=800.0 PL=0
MOVL C01517 V=800.0 PL=0
MOVL C01518 V=800.0 PL=0
MOVL C01519 V=800.0 PL=0
MOVL C01520 V=800.0 PL=0
MOVL C01521 V=800.0 PL=0
MOVL C01522 V=800.0 PL=0
MOVL C01523 V=800.0 PL=0
MOVL C01524 V=800.0 PL=0
MOVL C01525 V=800.0 PL=0
MOVL C01526 V=800.0 PL=0
MOVL C01527 V=800.0 PL=0
MOVL C01528 V=800.0 PL=0
MOVL C01529 V=800.0 PL=0
MOVL C01530 V=800.0 PL=0
MOVL C01531 V=800.0 PL=0
MOVL C01532 V=800.0 PL=0
MOVL C01533 V=800.0 PL=0
MOVL C01534 V=800.0 PL=0
MOVL C01535 V=800.0 PL=0
MOVL C01536 V=800.0 PL=0
MOVL C01537 V=800.0 PL=0
MOVL C01538 V=800.0 PL=0
MOVL C01539 V=800.0 PL=0
MOVL C01540 V=800.0 PL=0
MOVL C01541 V=800.0 PL=0
MOVL C01542 V=800.0 PL=0
MOVL C01543 V=800.0 PL=0
MOVL C01544 V=800.0 PL=0
MOVL C01545 V=800.0 PL=0
MOVL C01546 V=800.0 PL=0
MOVL C01547 V=800.0 PL=0
MOVL C01548 V=800.0 PL=0
MOVL C01549 V=800.0 PL=0
MOVL C01550 V=800.0 PL=0
MOVL C01551 V=800.0 PL=0
MOVL C01552 V=800.0 PL=0
MOVL C01553 V=800.0 PL=0
MOVL C01554 V=800.0 PL=0
MOVL C01555 V=800.0 PL=0
MOVL C01556 V=800.0 PL=0
MOVL C01557 V=800.0 PL=0
MOVL C01558 V=800.0 PL=0
MOVL C01559 V=800.0 PL=0
MOVL C01560 V=800.0 PL=0
MOVL C01561 V=800.0 PL=0
MOVL C01562 V=800.0 PL=0
MOVL C01563 V=800.0 PL=0
MOVL C01564 V=800.0 PL=0
MOVL C01565 V=800.0 PL=0
MOVL C01566 V=800.0 PL=0
MOVL C01567 V=800.0 PL=0
MOVL C01568 V=800.0 PL=0
MOVL C01569 V=800.0 PL=0
MOVL C01570 V=800.0 PL=0
MOVL C01571 V=800.0 PL=0
MOVL C01572 V=800.0 PL=0
MOVL C01573 V=800.0 PL=0
MOVL C01574 V=800.0 PL=0
MOVL C01575 V=800.0 PL=0
MOVL C01576 V=800.0 PL=0
MOVL C01577 V=800.0 PL=0
MOVL C01578 V=800.0 PL=0
MOVL C01579 V=800.0 PL=0
MOVL C01580 V=800.0 PL=0
MOVL C01581 V=800.0 PL=0
MOVL C01582 V=800.0 PL=0
MOVL C01583 V=800.0 PL=0
MOVL C01584 V=800.0 PL=0
MOVL C01585 V=800.0 PL=0
MOVL C01586 V=800.0 PL=0
MOVL C01587 V=800.0 PL=0
MOVL C01588 V=800.0 PL=0
MOVL C01589 V=800.0 PL=0
MOVL C01590 V=800.0 PL=0
MOVL C01591 V=800.0 PL=0
MOVL C01592 V=800.0 PL=0
MOVL C01593 V=800.0 PL=0
MOVL C01594 V=800.0 PL=0
MOVL C01595 V=800.0 PL=0
MOVL C01596 V=800.0 PL=0
MOVL C01597 V=800.0 PL=0
MOVL C01598 V=800.0 PL=0
MOVL C01599 V=800.0 PL=0
MOVL C01600 V=800.0 PL=0
MOVL C01601 V=800.0 PL=0
MOVL C01602 V=800.0 PL=0
MOVL C01603 V=800.0 PL=0
MOVL C01604 V=800.0 PL=0
MOVL C01605 V=800.0 PL=0
MOVL C01606 V=800.0 PL=0
MOVL C01607 V=800.0 PL=0
MOVL C01608 V=800.0 PL=0
MOVL C01609 V=800.0 PL=0
MOVL C01610 V=800.0 PL=0
MOVL C01611 V=800.0 PL=0
MOVL C01612 V=800.0 PL=0
MOVL C01613 V=800.0 PL=0
MOVL C01614 V=800.0 PL=0
MOVL C01615 V=800.0 PL=0
MOVL C01616 V=800.0 PL=0
MOVL C01617 V=800.0 PL=0
MOVL C01618 V=800.0 PL=0
MOVL C01619 V=800.0 PL=0
MOVL C01620 V=800.0 PL=0
MOVL C01621 V=800.0 PL=0
MOVL C01622 V=800.0 PL=0
MOVL C01623 V=800.0 PL=0
MOVL C01624 V=800.0 PL=0
MOVL C01625 V=800.0 PL=0
MOVL C01626 V=800.0 PL=0
MOVL C01627 V=800.0 PL=0
MOVL C01628 V=800.0 PL=0
MOVL C01629 V=800.0 PL=0
MOVL C01630 V=800.0 PL=0
MOVL C01631 V=800.0 PL=0
MOVL C01632 V=800.0 PL=0
MOVL C01633 V=800.0 PL=0
MOVL C01634 V=800.0 PL=0
MOVL C01635 V=800.0 PL=0
MOVL C01636 V=800.0 PL=0
MOVL C01637 V=800.0 PL=0
MOVL C01638 V=800.0 PL=0
MOVL C01639 V=800.0 PL=0
MOVL C01640 V=800.0 PL=0
MOVL C01641 V=800.0 PL=0
MOVL C01642 V=800.0 PL=0
MOVL C01643 V=800.0 PL=0
MOVL C01644 V=800.0 PL=0
MOVL C01645 V=800.0 PL=0
MOVL C01646 V=800.0 PL=0
MOVL C01647 V=800.0 PL=0
MOVL C01648 V=800.0 PL=0
MOVL C01649 V=800.0 PL=0
MOVL C01650 V=800.0 PL=0
MOVL C01651 V=800.0 PL=0
MOVL C01652 V=800.0 PL=0
MOVL C01653 V=800.0 PL=0
MOVL C01654 V=800.0 PL=0
MOVL C01655 V=800.0 PL=0
MOVL C01656 V=800.0 PL=0
MOVL C01657 V=800.0 PL=0
MOVL C01658 V=800.0 PL=0
MOVL C01659 V=800.0 PL=0
MOVL C01660 V=800.0 PL=0
MOVL C01661 V=800.0 PL=0
MOVL C01662 V=800.0 PL=0
MOVL C01663 V=800.0 PL=0
MOVL C01664 V=800.0 PL=0
MOVL C01665 V=800.0 PL=0
MOVL C01666 V=800.0 PL=0
MOVL C01667 V=800.0 PL=0
MOVL C01668 V=800.0 PL=0
MOVL C01669 V=800.0 PL=0
MOVL C01670 V=800.0 PL=0
MOVL C01671 V=800.0 PL=0
MOVL C01672 V=800.0 PL=0
MOVL C01673 V=800.0 PL=0
MOVL C01674 V=800.0 PL=0
MOVL C01675 V=800.0 PL=0
MOVL C01676 V=800.0 PL=0
MOVL C01677 V=800.0 PL=0
MOVL C01678 V=800.0 PL=0
MOVL C01679 V=800.0 PL=0
MOVL C01680 V=800.0 PL=0
MOVL C01681 V=800.0 PL=0
MOVL C01682 V=800.0 PL=0
MOVL C01683 V=800.0 PL=0
MOVL C01684 V=800.0 PL=0
MOVL C01685 V=800.0 PL=0
MOVL C01686 V=800.0 PL=0
MOVL C01687 V=800.0 PL=0
MOVL C01688 V=800.0 PL=0
MOVL C01689 V=800.0 PL=0
MOVL C01690 V=800.0 PL=0
MOVL C01691 V=800.0 PL=0
MOVL C01692 V=800.0 PL=0
MOVL C01693 V=800.0 PL=0
MOVL C01694 V=800.0 PL=0
MOVL C01695 V=800.0 PL=0
MOVL C01696 V=800.0 PL=0
MOVL C01697 V=800.0 PL=0
MOVL C01698 V=800.0 PL=0
MOVL C01699 V=800.0 PL=0
MOVL C01700 V=800.0 PL=0
MOVL C01701 V=800.0 PL=0
MOVL C01702 V=800.0 PL=0
MOVL C01703 V=800.0 PL=0
MOVL C01704 V=800.0 PL=0
MOVL C01705 V=800.0 PL=0
MOVL C01706 V=800.0 PL=0
MOVL C01707 V=800.0 PL=0
MOVL C01708 V=800.0 PL=0
MOVL C01709 V=800.0 PL=0
MOVL C01710 V=800.0 PL=0
MOVL C01711 V=800.0 PL=0
MOVL C01712 V=800.0 PL=0
MOVL C01713 V=800.0 PL=0
MOVL C01714 V=800.0 PL=0
MOVL C01715 V=800.0 PL=0
MOVL C01716 V=800.0 PL=0
MOVL C01717 V=800.0 PL=0
MOVL C01718 V=800.0 PL=0
MOVL C01719 V=800.0 PL=0
MOVL C01720 V=800.0 PL=0
MOVL C01721 V=800.0 PL=0
MOVL C01722 V=800.0 PL=0
MOVL C01723 V=800.0 PL=0
MOVL C01724 V=800.0 PL=0
MOVL C01725 V=800.0 PL=0
MOVL C01726 V=800.0 PL=0
MOVL C01727 V=800.0 PL=0
MOVL C01728 V=800.0 PL=0
MOVL C01729 V=800.0 PL=0
MOVL C01730 V=800.0 PL=0
MOVL C01731 V=800.0 PL=0
MOVL C01732 V=800.0 PL=0
MOVL C01733 V=800.0 PL=0
MOVL C01734 V=800.0 PL=0
MOVL C01735 V=800.0 PL=0
MOVL C01736 V=800.0 PL=0
MOVL C01737 V=800.0 PL=0
MOVL C01738 V=800.0 PL=0
MOVL C01739 V=800.0 PL=0
MOVL C01740 V=800.0 PL=0
MOVL C01741 V=800.0 PL=0
MOVL C01742 V=800.0 PL=0
MOVL C01743 V=800.0 PL=0
MOVL C01744 V=800.0 PL=0
MOVL C01745 V=800.0 PL=0
MOVL C01746 V=800.0 PL=0
MOVL C01747 V=800.0 PL=0
MOVL C01748 V=800.0 PL=0
MOVL C01749 V=800.0 PL=0
MOVL C01750 V=800.0 PL=0
MOVL C01751 V=800.0 PL=0
MOVL C01752 V=800.0 PL=0
MOVL C01753 V=800.0 PL=0
MOVL C01754 V=800.0 PL=0
MOVL C01755 V=800.0 PL=0
MOVL C01756 V=800.0 PL=0
MOVL C01757 V=800.0 PL=0
MOVL C01758 V=800.0 PL=0
MOVL C01759 V=800.0 PL=0
MOVL C01760 V=800.0 PL=0
MOVL C01761 V=800.0 PL=0
MOVL C01762 V=800.0 PL=0
MOVL C01763 V=800.0 PL=0
MOVL C01764 V=800.0 PL=0
MOVL C01765 V=800.0 PL=0
MOVL C01766 V=800.0 PL=0
MOVL C01767 V=800.0 PL=0
MOVL C01768 V=800.0 PL=0
MOVL C01769 V=800.0 PL=0
MOVL C01770 V=800.0 PL=0
MOVL C01771 V=800.0 PL=0
MOVL C01772 V=800.0 PL=0
MOVL C01773 V=800.0 PL=0
MOVL C01774 V=800.0 PL=0
MOVL C01775 V=800.0 PL=0
MOVL C01776 V=800.0 PL=0
MOVL C01777 V=800.0 PL=0
MOVL C01778 V=800.0 PL=0
MOVL C01779 V=800.0 PL=0
MOVL C01780 V=800.0 PL=0
MOVL C01781 V=800.0 PL=0
MOVL C01782 V=800.0 PL=0
MOVL C01783 V=800.0 PL=0
MOVL C01784 V=800.0 PL=0
MOVL C01785 V=800.0 PL=0
MOVL C01786 V=800.0 PL=0
MOVL C01787 V=800.0 PL=0
MOVL C01788 V=800.0 PL=0
MOVL C01789 V=800.0 PL=0
MOVL C01790 V=800.0 PL=0
MOVL C01791 V=800.0 PL=0
MOVL C01792 V=800.0 PL=0
MOVL C01793 V=800.0 PL=0
MOVL C01794 V=800.0 PL=0
MOVL C01795 V=800.0 PL=0
MOVL C01796 V=800.0 PL=0
MOVL C01797 V=800.0 PL=0
MOVL C01798 V=800.0 PL=0
MOVL C01799 V=800.0 PL=0
MOVL C01800 V=800.0 PL=0
MOVL C01801 V=800.0 PL=0
MOVL C01802 V=800.0 PL=0
MOVL C01803 V=800.0 PL=0
MOVL C01804 V=800.0 PL=0
MOVL C01805 V=800.0 PL=0
MOVL C01806 V=800.0 PL=0
MOVL C01807 V=800.0 PL=0
MOVL C01808 V=800.0 PL=0
MOVL C01809 V=800.0 PL=0
MOVL C01810 V=800.0 PL=0
MOVL C01811 V=800.0 PL=0
MOVL C01812 V=800.0 PL=0
MOVL C01813 V=800.0 PL=0
MOVL C01814 V=800.0 PL=0
MOVL C01815 V=800.0 PL=0
MOVL C01816 V=800.0 PL=0
MOVL C01817 V=800.0 PL=0
MOVL C01818 V=800.0 PL=0
MOVL C01819 V=800.0 PL=0
MOVL C01820 V=800.0 PL=0
MOVL C01821 V=800.0 PL=0
MOVL C01822 V=800.0 PL=0
MOVL C01823 V=800.0 PL=0
MOVL C01824 V=800.0 PL=0
MOVL C01825 V=800.0 PL=0
MOVL C01826 V=800.0 PL=0
MOVL C01827 V=800.0 PL=0
MOVL C01828 V=800.0 PL=0
MOVL C01829 V=800.0 PL=0
MOVL C01830 V=800.0 PL=0
MOVL C01831 V=800.0 PL=0
MOVL C01832 V=800.0 PL=0
MOVL C01833 V=800.0 PL=0
MOVL C01834 V=800.0 PL=0
MOVL C01835 V=800.0 PL=0
MOVL C01836 V=800.0 PL=0
MOVL C01837 V=800.0 PL=0
MOVL C01838 V=800.0 PL=0
MOVL C01839 V=800.0 PL=0
MOVL C01840 V=800.0 PL=0
MOVL C01841 V=800.0 PL=0
MOVL C01842 V=800.0 PL=0
MOVL C01843 V=800.0 PL=0
MOVL C01844 V=800.0 PL=0
MOVL C01845 V=800.0 PL=0
MOVL C01846 V=800.0 PL=0
MOVL C01847 V=800.0 PL=0
MOVL C01848 V=800.0 PL=0
MOVL C01849 V=800.0 PL=0
MOVL C01850 V=800.0 PL=0
MOVL C01851 V=800.0 PL=0
MOVL C01852 V=800.0 PL=0
MOVL C01853 V=800.0 PL=0
MOVL C01854 V=800.0 PL=0
MOVL C01855 V=800.0 PL=0
MOVL C01856 V=800.0 PL=0
MOVL C01857 V=800.0 PL=0
MOVL C01858 V=800.0 PL=0
MOVL C01859 V=800.0 PL=0
MOVL C01860 V=800.0 PL=0
MOVL C01861 V=800.0 PL=0
MOVL C01862 V=800.0 PL=0
MOVL C01863 V=800.0 PL=0
MOVL C01864 V=800.0 PL=0
MOVL C01865 V=800.0 PL=0
MOVL C01866 V=800.0 PL=0
MOVL C01867 V=800.0 PL=0
MOVL C01868 V=800.0 PL=0
MOVL C01869 V=800.0 PL=0
MOVL C01870 V=800.0 PL=0
MOVL C01871 V=800.0 PL=0
MOVL C01872 V=800.0 PL=0
MOVL C01873 V=800.0 PL=0
MOVL C01874 V=800.0 PL=0
MOVL C01875 V=800.0 PL=0
MOVL C01876 V=800.0 PL=0
MOVL C01877 V=800.0 PL=0
MOVL C01878 V=800.0 PL=0
MOVL C01879 V=800.0 PL=0
MOVL C01880 V=800.0 PL=0
MOVL C01881 V=800.0 PL=0
MOVL C01882 V=800.0 PL=0
MOVL C01883 V=800.0 PL=0
MOVL C01884 V=800.0 PL=0
MOVL C01885 V=800.0 PL=0
MOVL C01886 V=800.0 PL=0
MOVL C01887 V=800.0 PL=0
MOVL C01888 V=800.0 PL=0
MOVL C01889 V=800.0 PL=0
MOVL C01890 V=800.0 PL=0
MOVL C01891 V=800.0 PL=0
MOVL C01892 V=800.0 PL=0
MOVL C01893 V=800.0 PL=0
MOVL C01894 V=800.0 PL=0
MOVL C01895 V=800.0 PL=0
MOVL C01896 V=800.0 PL=0
MOVL C01897 V=800.0 PL=0
MOVL C01898 V=800.0 PL=0
MOVL C01899 V=800.0 PL=0
MOVL C01900 V=800.0 PL=0
MOVL C01901 V=800.0 PL=0
MOVL C01902 V=800.0 PL=0
MOVL C01903 V=800.0 PL=0
MOVL C01904 V=800.0 PL=0
MOVL C01905 V=800.0 PL=0
MOVL C01906 V=800.0 PL=0
MOVL C01907 V=800.0 PL=0
MOVL C01908 V=800.0 PL=0
MOVL C01909 V=800.0 PL=0
MOVL C01910 V=800.0 PL=0
MOVL C01911 V=800.0 PL=0
MOVL C01912 V=800.0 PL=0
MOVL C01913 V=800.0 PL=0
MOVL C01914 V=800.0 PL=0
MOVL C01915 V=800.0 PL=0
MOVL C01916 V=800.0 PL=0
MOVL C01917 V=800.0 PL=0
MOVL C01918 V=800.0 PL=0
MOVL C01919 V=800.0 PL=0
MOVL C01920 V=800.0 PL=0
MOVL C01921 V=800.0 PL=0
MOVL C01922 V=800.0 PL=0
MOVL C01923 V=800.0 PL=0
MOVL C01924 V=800.0 PL=0
MOVL C01925 V=800.0 PL=0
MOVL C01926 V=800.0 PL=0
MOVL C01927 V=800.0 PL=0
MOVL C01928 V=800.0 PL=0
MOVL C01929 V=800.0 PL=0
MOVL C01930 V=800.0 PL=0
MOVL C01931 V=800.0 PL=0
MOVL C01932 V=800.0 PL=0
MOVL C01933 V=800.0 PL=0
MOVL C01934 V=800.0 PL=0
MOVL C01935 V=800.0 PL=0
MOVL C01936 V=800.0 PL=0
MOVL C01937 V=800.0 PL=0
MOVL C01938 V=800.0 PL=0
MOVL C01939 V=800.0 PL=0
MOVL C01940 V=800.0 PL=0
MOVL C01941 V=800.0 PL=0
MOVL C01942 V=800.0 PL=0
MOVL C01943 V=800.0 PL=0
MOVL C01944 V=800.0 PL=0
MOVL C01945 V=800.0 PL=0
MOVL C01946 V=800.0 PL=0
MOVL C01947 V=800.0 PL=0
MOVL C01948 V=800.0 PL=0
MOVL C01949 V=800.0 PL=0
MOVL C01950 V=800.0 PL=0
MOVL C01951 V=800.0 PL=0
MOVL C01952 V=800.0 PL=0
MOVL C01953 V=800.0 PL=0
MOVL C01954 V=800.0 PL=0
MOVL C01955 V=800.0 PL=0
MOVL C01956 V=800.0 PL=0
MOVL C01957 V=800.0 PL=0
MOVL C01958 V=800.0 PL=0
MOVL C01959 V=800.0 PL=0
MOVL C01960 V=800.0 PL=0
MOVL C01961 V=800.0 PL=0
MOVL C01962 V=800.0 PL=0
MOVL C01963 V=800.0 PL=0
MOVL C01964 V=800.0 PL=0
MOVL C01965 V=800.0 PL=0
MOVL C01966 V=800.0 PL=0
MOVL C01967 V=800.0 PL=0
MOVL C01968 V=800.0 PL=0
MOVL C01969 V=800.0 PL=0
MOVL C01970 V=800.0 PL=0
MOVL C01971 V=800.0 PL=0
MOVL C01972 V=800.0 PL=0
MOVL C01973 V=800.0 PL=0
MOVL C01974 V=800.0 PL=0
MOVL C01975 V=800.0 PL=0
MOVL C01976 V=800.0 PL=0
MOVL C01977 V=800.0 PL=0
MOVL C01978 V=800.0 PL=0
MOVL C01979 V=800.0 PL=0
MOVL C01980 V=800.0 PL=0
MOVL C01981 V=800.0 PL=0
MOVL C01982 V=800.0 PL=0
MOVL C01983 V=800.0 PL=0
MOVL C01984 V=800.0 PL=0
MOVL C01985 V=800.0 PL=0
MOVL C01986 V=800.0 PL=0
MOVL C01987 V=800.0 PL=0
MOVL C01988 V=800.0 PL=0
MOVL C01989 V=800.0 PL=0
MOVL C01990 V=800.0 PL=0
MOVL C01991 V=800.0 PL=0
MOVL C01992 V=800.0 PL=0
MOVL C01993 V=800.0 PL=0
MOVL C01994 V=800.0 PL=0
MOVL C01995 V=800.0 PL=0
MOVL C01996 V=800.0 PL=0
MOVL C01997 V=800.0 PL=0
MOVL C01998 V=800.0 PL=0
MOVL C01999 V=800.0 PL=0
MOVL C02000 V=800.0 PL=0
MOVL C02001 V=800.0 PL=0
MOVL C02002 V=800.0 PL=0
MOVL C02003 V=800.0 PL=0
MOVL C02004 V=800.0 PL=0
MOVL C02005 V=800.0 PL=0
MOVL C02006 V=800.0 PL=0
MOVL C02007 V=800.0 PL=0
MOVL C02008 V=800.0 PL=0
MOVL C02009 V=800.0 PL=0
MOVL C02010 V=800.0 PL=0
MOVL C02011 V=800.0 PL=0
MOVL C02012 V=800.0 PL=0
MOVL C02013 V=800.0 PL=0
MOVL C02014 V=800.0 PL=0
MOVL C02015 V=800.0 PL=0
MOVL C02016 V=800.0 PL=0
MOVL C02017 V=800.0 PL=0
MOVL C02018 V=800.0 PL=0
MOVL C02019 V=800.0 PL=0
MOVL C02020 V=800.0 PL=0
MOVL C02021 V=800.0 PL=0
MOVL C02022 V=800.0 PL=0
MOVL C02023 V=800.0 PL=0
MOVL C02024 V=800.0 PL=0
MOVL C02025 V=800.0 PL=0
MOVL C02026 V=800.0 PL=0
MOVL C02027 V=800.0 PL=0
MOVL C02028 V=800.0 PL=0
MOVL C02029 V=800.0 PL=0
MOVL C02030 V=800.0 PL=0
MOVL C02031 V=800.0 PL=0
MOVL C02032 V=800.0 PL=0
MOVL C02033 V=800.0 PL=0
MOVL C02034 V=800.0 PL=0
MOVL C02035 V=800.0 PL=0
MOVL C02036 V=800.0 PL=0
MOVL C02037 V=800.0 PL=0
MOVL C02038 V=800.0 PL=0
MOVL C02039 V=800.0 PL=0
MOVL C02040 V=800.0 PL=0
